Omron Sysmac Studio project 17-701_20171123 (Sysmac Studio 1.19.0.13, StandardProject)

# Controller new_Controller_0: NJ101-1000 version 1.13
Units and slaves: 電源 : NJ-Px3001; CPU : NJ101-1000; 0 : CJ1W-ID211 (J01); 1 : CJ1W-OD211 (J02)
Task PrimaryTask (priority 4, period or condition 2000): prIndexDataChange, prIndex, prError, prSystemInit, prError_S0, prError_S1, prError_S2, prError_S4, prError_S6, prError_S8, prError_S10, prError_S11, prError_S13, prError_S15, prStation1, prStation1_Robot, prStation1_PanelLoad, prStation1_FeedPanelLoad, prStation1_PanelUnLoad, prStation1_FeedPanelUnLoad, prStation2, prStation4, prStation4_TH, prStation4_PanelLoad, prStation4_PanelUnLoad, prStation5, prStation6, prStation7, prStation8, prStation8_CCD, prStation8_ChangeJig, prStation9, prStation10, prStation11, prStation13, prStation15, prStation16, prFeedAndSupplier, prNGCount

TYPE stIndexData : STRUCT
    FinishFlag : ARRAY[0..19] OF BOOL;
    OKFlag : ARRAY[0..19] OF BOOL;
    NGFlag : ARRAY[0..19] OF BOOL;
    ErrorLog : ARRAY[0..19] OF INT;
END_STRUCT END_TYPE

VAR_GLOBAL
    LS_S1_Load_PanelUpDown1Back : BOOL;  (* at ECAT://node#[1,1]/Input Bit 16 bits/Input Bit 00; published *)
    LS_S1_Load_PanelUpDown1Out : BOOL;  (* at ECAT://node#[1,1]/Input Bit 16 bits/Input Bit 01; published *)
    LS_S1_Load_PanelUpDown2Back : BOOL;  (* at ECAT://node#[1,1]/Input Bit 16 bits/Input Bit 02; published *)
    LS_S1_Load_PanelUpDown2Out : BOOL;  (* at ECAT://node#[1,1]/Input Bit 16 bits/Input Bit 03; published *)
    LS_S1_Load_PanelClip1Back : BOOL;  (* at ECAT://node#[1,1]/Input Bit 16 bits/Input Bit 04; published *)
    LS_S1_Load_PanelClip1Out : BOOL;  (* at ECAT://node#[1,1]/Input Bit 16 bits/Input Bit 05; published *)
    LS_S1_Load_PanelClip2Back : BOOL;  (* at ECAT://node#[1,1]/Input Bit 16 bits/Input Bit 06; published *)
    LS_S1_Load_PanelClip2Out : BOOL;  (* at ECAT://node#[1,1]/Input Bit 16 bits/Input Bit 07; published *)
    LS_S1_Load_FixClipBack : BOOL;  (* at ECAT://node#[1,1]/Input Bit 16 bits/Input Bit 08; published *)
    LS_S1_Load_FixClipOut : BOOL;  (* at ECAT://node#[1,1]/Input Bit 16 bits/Input Bit 09; published *)
    LS_S1_Load_AlignmentClipBack : BOOL;  (* at ECAT://node#[1,1]/Input Bit 16 bits/Input Bit 10; published *)
    LS_S1_Load_AlignmentClipOut : BOOL;  (* at ECAT://node#[1,1]/Input Bit 16 bits/Input Bit 11; published *)
    LS_S1_Load_ConveyorClip1Back : BOOL;  (* at ECAT://node#[1,1]/Input Bit 16 bits/Input Bit 12; published *)
    LS_S1_Load_ConveyorClip1Out : BOOL;  (* at ECAT://node#[1,1]/Input Bit 16 bits/Input Bit 13; published *)
    LS_S1_Load_ConveyorClip2Back : BOOL;  (* at ECAT://node#[1,1]/Input Bit 16 bits/Input Bit 14; published *)
    LS_S1_Load_ConveyorClip2Out : BOOL;  (* at ECAT://node#[1,1]/Input Bit 16 bits/Input Bit 15; published *)
    LS_S1_Load_UpDownBack : BOOL;  (* at ECAT://node#[1,2]/Input Bit 16 bits/Input Bit 00; published *)
    LS_S1_Load_UpDownOut : BOOL;  (* at ECAT://node#[1,2]/Input Bit 16 bits/Input Bit 01; published *)
    LS_S1_UnLoad_UpDownBack : BOOL;  (* at ECAT://node#[1,2]/Input Bit 16 bits/Input Bit 02; published *)
    LS_S1_UnLoad_UpDownOut : BOOL;  (* at ECAT://node#[1,2]/Input Bit 16 bits/Input Bit 03; published *)
    LS_S1_UnLoad_ConveyorClip1Back : BOOL;  (* at ECAT://node#[1,2]/Input Bit 16 bits/Input Bit 04; published *)
    LS_S1_UnLoad_ConveyorClip1Out : BOOL;  (* at ECAT://node#[1,2]/Input Bit 16 bits/Input Bit 05; published *)
    LS_S1_UnLoad_ConveyorClip2Back : BOOL;  (* at ECAT://node#[1,2]/Input Bit 16 bits/Input Bit 06; published *)
    LS_S1_UnLoad_ConveyorClip2Out : BOOL;  (* at ECAT://node#[1,2]/Input Bit 16 bits/Input Bit 07; published *)
    LS_S1_UnLoad_FixClipBack : BOOL;  (* at ECAT://node#[1,2]/Input Bit 16 bits/Input Bit 08; published *)
    LS_S1_UnLoad_FixClipOut : BOOL;  (* at ECAT://node#[1,2]/Input Bit 16 bits/Input Bit 09; published *)
    LS_S1_UnLoad_AlignmentClipBack : BOOL;  (* at ECAT://node#[1,2]/Input Bit 16 bits/Input Bit 10; published *)
    LS_S1_UnLoad_AlignmentClipOut : BOOL;  (* at ECAT://node#[1,2]/Input Bit 16 bits/Input Bit 11; published *)
    LS_S1_UnLoad_PanelClip1Back : BOOL;  (* at ECAT://node#[1,2]/Input Bit 16 bits/Input Bit 12; published *)
    LS_S1_UnLoad_PanelClip1Out : BOOL;  (* at ECAT://node#[1,2]/Input Bit 16 bits/Input Bit 13; published *)
    LS_S1_UnLoad_PanelClip2Back : BOOL;  (* at ECAT://node#[1,2]/Input Bit 16 bits/Input Bit 14; published *)
    LS_S1_UnLoad_PanelClip2Out : BOOL;  (* at ECAT://node#[1,2]/Input Bit 16 bits/Input Bit 15; published *)
    LS_S1_UnLoad_PanelUpDown1Back : BOOL;  (* at ECAT://node#[1,3]/Input Bit 16 bits/Input Bit 00; published *)
    LS_S1_UnLoad_PanelUpDown1Out : BOOL;  (* at ECAT://node#[1,3]/Input Bit 16 bits/Input Bit 01; published *)
    LS_S1_UnLoad_PanelUpDown2Back : BOOL;  (* at ECAT://node#[1,3]/Input Bit 16 bits/Input Bit 02; published *)
    LS_S1_UnLoad_PanelUpDown2Out : BOOL;  (* at ECAT://node#[1,3]/Input Bit 16 bits/Input Bit 03; published *)
    SNR_S1_Load_Full : BOOL;  (* 出盤缺盤檢知; at ECAT://node#[1,3]/Input Bit 16 bits/Input Bit 08; published *)
    SNR_S1_UnLoad_Full : BOOL;  (* 收盤滿盤檢知; at ECAT://node#[1,3]/Input Bit 16 bits/Input Bit 09; published *)
    SNR_S1_Load_Feed : BOOL;  (* 下移載出盤檢知; at ECAT://node#[1,3]/Input Bit 16 bits/Input Bit 10; published *)
    SNR_S1_UnLoad_Feed : BOOL;  (* 下移載收盤檢知; at ECAT://node#[1,3]/Input Bit 16 bits/Input Bit 11; published *)
    SNR_S1_Load_PanelFeed : BOOL;  (* 出盤下盤處檢知; at ECAT://node#[1,3]/Input Bit 16 bits/Input Bit 12; published *)
    SNR_S1_Load_PanelClip : BOOL;  (* 出盤夾盤處檢知; at ECAT://node#[1,3]/Input Bit 16 bits/Input Bit 13; published *)
    SNR_S1_UnLoad_PanelFeed : BOOL;  (* 收盤上盤處檢知; at ECAT://node#[1,3]/Input Bit 16 bits/Input Bit 14; published *)
    SNR_S1_UnLoad_PanelClip : BOOL;  (* 收盤夾盤處檢知; at ECAT://node#[1,3]/Input Bit 16 bits/Input Bit 15; published *)
    SOL_S1_Load_PanelUpDown1Back : BOOL;  (* at ECAT://node#[1,4]/Output Bit 16 bits/Output Bit 00; published *)
    SOL_S1_Load_PanelUpDown1Out : BOOL;  (* at ECAT://node#[1,4]/Output Bit 16 bits/Output Bit 01; published *)
    SOL_S1_Load_PanelUpDown2Back : BOOL;  (* at ECAT://node#[1,4]/Output Bit 16 bits/Output Bit 02; published *)
    SOL_S1_Load_PanelUpDown2Out : BOOL;  (* at ECAT://node#[1,4]/Output Bit 16 bits/Output Bit 03; published *)
    SOL_S1_Load_PanelClip : BOOL;  (* at ECAT://node#[1,4]/Output Bit 16 bits/Output Bit 04; published *)
    SOL_S1_Load_FixClip : BOOL;  (* at ECAT://node#[1,4]/Output Bit 16 bits/Output Bit 05; published *)
    SOL_S1_Load_AlignmentClip : BOOL;  (* at ECAT://node#[1,4]/Output Bit 16 bits/Output Bit 06; published *)
    SOL_S1_Load_ConveyorClip : BOOL;  (* at ECAT://node#[1,4]/Output Bit 16 bits/Output Bit 07; published *)
    SOL_S1_Load_UpDown : BOOL;  (* at ECAT://node#[1,4]/Output Bit 16 bits/Output Bit 08; published *)
    RY_S1_Load_FixSpeedMotor : BOOL;  (* at ECAT://node#[1,4]/Output Bit 16 bits/Output Bit 09; published *)
    RY_S1_UnLoad_FixSpeedMotor : BOOL;  (* at ECAT://node#[1,4]/Output Bit 16 bits/Output Bit 10; published *)
    RY_S1_Load_VariableSpeedMotor : BOOL;  (* at ECAT://node#[1,4]/Output Bit 16 bits/Output Bit 11; published *)
    RY_S1_UnLoad_VariableSpeedMotor : BOOL;  (* at ECAT://node#[1,4]/Output Bit 16 bits/Output Bit 12; published *)
    RY_S1_Center_VariableSpeedMotor : BOOL;  (* at ECAT://node#[1,4]/Output Bit 16 bits/Output Bit 13; published *)
    SOL_S1_UnLoad_PanelUpDown1Back : BOOL;  (* at ECAT://node#[1,8]/Output Bit 16 bits/Output Bit 00; published *)
    SOL_S1_UnLoad_PanelUpDown1Out : BOOL;  (* at ECAT://node#[1,8]/Output Bit 16 bits/Output Bit 01; published *)
    SOL_S1_UnLoad_PanelUpDown2Back : BOOL;  (* at ECAT://node#[1,8]/Output Bit 16 bits/Output Bit 02; published *)
    SOL_S1_UnLoad_PanelUpDown2Out : BOOL;  (* at ECAT://node#[1,8]/Output Bit 16 bits/Output Bit 03; published *)
    SOL_S1_UnLoad_PanelClip : BOOL;  (* at ECAT://node#[1,8]/Output Bit 16 bits/Output Bit 04; published *)
    SOL_S1_UnLoad_FixClip : BOOL;  (* at ECAT://node#[1,8]/Output Bit 16 bits/Output Bit 05; published *)
    SOL_S1_UnLoad_AlignmentClip : BOOL;  (* at ECAT://node#[1,8]/Output Bit 16 bits/Output Bit 06; published *)
    SOL_S1_UnLoad_ConveyorClip : BOOL;  (* at ECAT://node#[1,8]/Output Bit 16 bits/Output Bit 07; published *)
    SOL_S1_UnLoad_UpDown : BOOL;  (* at ECAT://node#[1,8]/Output Bit 16 bits/Output Bit 08; published *)
    YAMAHA_Unload_OKStart : BOOL;  (* at ECAT://node#[1,5]/Output Bit 16 bits/Output Bit 00; published *)
    YAMAHA_Unload_NGStart : BOOL;  (* at ECAT://node#[1,5]/Output Bit 16 bits/Output Bit 01; published *)
    YAMAHA_Load_Start : BOOL;  (* at ECAT://node#[1,5]/Output Bit 16 bits/Output Bit 02; published *)
    YAMAHA_UnLoad_Ready : BOOL;  (* at ECAT://node#[1,5]/Output Bit 16 bits/Output Bit 03; published *)
    YAMAHA_Load_Ready : BOOL;  (* at ECAT://node#[1,5]/Output Bit 16 bits/Output Bit 04; published *)
    YAMAHA_Error_SOL_Clip : BOOL;  (* at ECAT://node#[1,6]/Input Bit 16 bits/Input Bit 00; published *)
    YAMAHA_Unload_Finish : BOOL;  (* at ECAT://node#[1,6]/Input Bit 16 bits/Input Bit 01; published *)
    YAMAHA_Load_Finish : BOOL;  (* at ECAT://node#[1,6]/Input Bit 16 bits/Input Bit 02; published *)
    YAMAHA_Unload_ChangePanelStart : BOOL;  (* at ECAT://node#[1,6]/Input Bit 16 bits/Input Bit 03; published *)
    YAMAHA_Load_ChangePanelStart : BOOL;  (* at ECAT://node#[1,6]/Input Bit 16 bits/Input Bit 04; published *)
    YAMAHA_ORG : BOOL;  (* at ECAT://node#[1,6]/Input Bit 16 bits/Input Bit 05; published *)
    YAMAHA_S_Enable : BOOL;  (* at ECAT://node#[1,5]/Output Bit 16 bits/Output Bit 08; published *)
    YAMAHA_S_Control : BOOL;  (* at ECAT://node#[1,5]/Output Bit 16 bits/Output Bit 09; published *)
    YAMAHA_S_Stop : BOOL;  (* at ECAT://node#[1,5]/Output Bit 16 bits/Output Bit 10; published *)
    YAMAHA_S_AutoRun : BOOL;  (* at ECAT://node#[1,5]/Output Bit 16 bits/Output Bit 11; published *)
    YAMAHA_S_INCHome : BOOL;  (* at ECAT://node#[1,5]/Output Bit 16 bits/Output Bit 12; published *)
    YAMAHA_S_ProgramReset : BOOL;  (* at ECAT://node#[1,5]/Output Bit 16 bits/Output Bit 13; published *)
    YAMAHA_S_AlarmReset : BOOL;  (* at ECAT://node#[1,5]/Output Bit 16 bits/Output Bit 14; published *)
    YAMAHA_S_ABSHome : BOOL;  (* at ECAT://node#[1,5]/Output Bit 16 bits/Output Bit 15; published *)
    YAMAHA_S_State_CPUOK : BOOL;  (* at ECAT://node#[1,6]/Input Bit 16 bits/Input Bit 08; published *)
    YAMAHA_S_State_AutoMode : BOOL;  (* at ECAT://node#[1,6]/Input Bit 16 bits/Input Bit 09; published *)
    YAMAHA_S_State_Homed : BOOL;  (* at ECAT://node#[1,6]/Input Bit 16 bits/Input Bit 10; published *)
    YAMAHA_S_State_RobotProgramRun : BOOL;  (* at ECAT://node#[1,6]/Input Bit 16 bits/Input Bit 11; published *)
    YAMAHA_S_State_ProgramReset : BOOL;  (* at ECAT://node#[1,6]/Input Bit 16 bits/Input Bit 12; published *)
    YAMAHA_S_State_Warring : BOOL;  (* at ECAT://node#[1,6]/Input Bit 16 bits/Input Bit 13; published *)
    YAMAHA_S_State_Enable : BOOL;  (* at ECAT://node#[1,6]/Input Bit 16 bits/Input Bit 14; published *)
    YAMAHA_S_State_Alarm : BOOL;  (* at ECAT://node#[1,6]/Input Bit 16 bits/Input Bit 15; published *)
    SNR_S1_Door1 : BOOL;  (* at ECAT://node#[1,3]/Input Bit 16 bits/Input Bit 04; published *)
    SNR_S1_Door2 : BOOL;  (* at ECAT://node#[1,3]/Input Bit 16 bits/Input Bit 05; published *)
    SNR_S1_Door3 : BOOL;  (* at ECAT://node#[1,3]/Input Bit 16 bits/Input Bit 06; published *)
    SNR_S1_Door4 : BOOL;  (* at ECAT://node#[1,3]/Input Bit 16 bits/Input Bit 07; published *)
    LS_S4_Load_PanelUpDown1Back : BOOL;  (* published *)
    LS_S4_Load_PanelUpDown1Out : BOOL;  (* published *)
    LS_S4_Load_PanelUpDown2Back : BOOL;  (* published *)
    LS_S4_Load_PanelUpDown2Out : BOOL;  (* published *)
    LS_S4_Load_PanelClip1Back : BOOL;  (* published *)
    LS_S4_Load_PanelClip1Out : BOOL;  (* published *)
    LS_S4_Load_PanelClip2Back : BOOL;  (* published *)
    LS_S4_Load_PanelClip2Out : BOOL;  (* published *)
    LS_S4_UnLoad_PanelUpDown1Back : BOOL;  (* published *)
    LS_S4_UnLoad_PanelUpDown1Out : BOOL;  (* published *)
    LS_S4_UnLoad_PanelUpDown2Back : BOOL;  (* published *)
    LS_S4_UnLoad_PanelUpDown2Out : BOOL;  (* published *)
    LS_S4_UnLoad_PanelClip1Back : BOOL;  (* published *)
    LS_S4_UnLoad_PanelClip1Out : BOOL;  (* published *)
    LS_S4_UnLoad_PanelClip2Back : BOOL;  (* published *)
    LS_S4_UnLoad_PanelClip2Out : BOOL;  (* published *)
    LS_S4_Center_UpDownBack : BOOL;  (* published *)
    LS_S4_Center_UpDownOut : BOOL;  (* published *)
    LS_S4_Center_ClipBack : BOOL;  (* published *)
    LS_S4_Center_ClipOut : BOOL;  (* published *)
    SNR_S4_Load_Feed : BOOL;  (* published *)
    SNR_S4_UnLoad_Feed : BOOL;  (* published *)
    SNR_S4_Load_Full : BOOL;  (* published *)
    SNR_S4_UnLoad_Full : BOOL;  (* published *)
    SOL_S4_Load_PanelUpDown1Back : BOOL;  (* published *)
    SOL_S4_Load_PanelUpDown1Out : BOOL;  (* published *)
    SOL_S4_Load_PanelUpDown2Back : BOOL;  (* published *)
    SOL_S4_Load_PanelUpDown2Out : BOOL;  (* published *)
    SOL_S4_Load_PanelClip : BOOL;  (* published *)
    SOL_S4_UnLoad_PanelUpDown1Back : BOOL;  (* published *)
    SOL_S4_UnLoad_PanelUpDown1Out : BOOL;  (* published *)
    SOL_S4_UnLoad_PanelUpDown2Back : BOOL;  (* published *)
    SOL_S4_UnLoad_PanelUpDown2Out : BOOL;  (* published *)
    SOL_S4_UnLoad_PanelClip : BOOL;  (* published *)
    SOL_S4_Center_UpDown : BOOL;  (* published *)
    SOL_S4_Center_Clip : BOOL;  (* published *)
    SOL_S2_UpDown : BOOL;  (* published *)
    SOL_S4_MoveBack : BOOL;  (* published *)
    SOL_S4_MoveOut : BOOL;  (* published *)
    SOL_S4_UpDown : BOOL;  (* published *)
    SOL_S4_Clip : BOOL;  (* published *)
    SOL_S4_THMoveBack : BOOL;  (* published *)
    SOL_S4_THMoveOut : BOOL;  (* published *)
    SOL_S6_MoveBack : BOOL;  (* published *)
    SOL_S6_MoveOut : BOOL;  (* published *)
    SOL_S6_UpDown : BOOL;  (* published *)
    SOL_S6_TH : BOOL;  (* published *)
    SOL_S8_MoveBack : BOOL;  (* published *)
    SOL_S8_MoveOut : BOOL;  (* published *)
    SOL_S8_UpDown : BOOL;  (* published *)
    SOL_S8_FixMove : BOOL;  (* published *)
    SOL_S8_Fix : BOOL;  (* published *)
    SOL_S8_TH : BOOL;  (* published *)
    SOL_S8_Turn : BOOL;  (* published *)
    SOL_S8_Clip : BOOL;  (* published *)
    SOL_S10_MoveBack : BOOL;  (* published *)
    SOL_S10_MoveOut : BOOL;  (* published *)
    SOL_S10_UpDown : BOOL;  (* published *)
    SOL_S10_ClipF : BOOL;  (* published *)
    SOL_S10_ClipR : BOOL;  (* published *)
    SOL_S10_TH : BOOL;  (* published *)
    SOL_S10_Turn : BOOL;  (* published *)
    SOL_S11_UpDown : BOOL;  (* published *)
    SOL_S13_UpDown : BOOL;  (* published *)
    SOL_S15_UpDown : BOOL;  (* published *)
    SOL_S6_Vacuum : BOOL;  (* published *)
    SOL_S6_Break : BOOL;  (* published *)
    SOL_S8_VacuumF : BOOL;  (* published *)
    SOL_S8_BreakF : BOOL;  (* published *)
    SOL_S8_VacuumR : BOOL;  (* published *)
    SOL_S8_BreakR : BOOL;  (* published *)
    RY_S6_Full : BOOL;  (* published *)
    RY_S6_Feed : BOOL;  (* published *)
    RY_S8_Full : BOOL;  (* published *)
    RY_S8_Feed : BOOL;  (* published *)
    RY_S10_Full : BOOL;  (* published *)
    RY_S10_Feed : BOOL;  (* published *)
    LS_S2_UpDownBack : BOOL;  (* published *)
    LS_S2_UpDownOut : BOOL;  (* published *)
    LS_S4_MoveBack : BOOL;  (* published *)
    LS_S4_MoveOut : BOOL;  (* published *)
    LS_S4_UpDownBack : BOOL;  (* published *)
    LS_S4_UpDownOut : BOOL;  (* published *)
    LS_S4_ClipBack : BOOL;  (* published *)
    LS_S4_ClipOut : BOOL;  (* published *)
    LS_S4_THMoveBack : BOOL;  (* published *)
    LS_S4_THMoveOut : BOOL;  (* published *)
    LS_S6_MoveBack : BOOL;  (* published *)
    LS_S6_MoveOut : BOOL;  (* published *)
    LS_S6_UpDownBack : BOOL;  (* published *)
    LS_S6_UpDownOut : BOOL;  (* published *)
    LS_S6_THBack : BOOL;  (* published *)
    LS_S6_THOut : BOOL;  (* published *)
    LS_S8_MoveBack : BOOL;  (* published *)
    LS_S8_MoveOut : BOOL;  (* published *)
    LS_S8_UpDownBack : BOOL;  (* published *)
    LS_S8_UpDownOut : BOOL;  (* published *)
    LS_S8_FixMoveBack : BOOL;  (* published *)
    LS_S8_FixMoveOut : BOOL;  (* published *)
    LS_S8_FixBack : BOOL;  (* published *)
    LS_S8_FixOut : BOOL;  (* published *)
    LS_S8_THBack : BOOL;  (* published *)
    LS_S8_THOut : BOOL;  (* published *)
    LS_S8_TurnBack : BOOL;  (* published *)
    LS_S8_TurnOut : BOOL;  (* published *)
    LS_S8_ClipBack : BOOL;  (* published *)
    LS_S8_ClipOut : BOOL;  (* published *)
    LS_S10_MoveBack : BOOL;  (* published *)
    LS_S10_MoveOut : BOOL;  (* published *)
    LS_S10_UpDownBack : BOOL;  (* published *)
    LS_S10_UpDownOut : BOOL;  (* published *)
    LS_S10_ClipFBack : BOOL;  (* published *)
    LS_S10_ClipFOut : BOOL;  (* published *)
    LS_S10_ClipRBack : BOOL;  (* published *)
    LS_S10_ClipROut : BOOL;  (* published *)
    LS_S10_THBack : BOOL;  (* published *)
    LS_S10_THOut : BOOL;  (* published *)
    LS_S10_TurnBack : BOOL;  (* published *)
    LS_S10_TurnOut : BOOL;  (* published *)
    LS_S11_UpDownBack : BOOL;  (* published *)
    LS_S11_UpDownOut : BOOL;  (* published *)
    LS_S13_UpDownBack : BOOL;  (* published *)
    LS_S13_UpDownOut : BOOL;  (* published *)
    LS_S15_UpDownBack : BOOL;  (* published *)
    LS_S15_UpDownOut : BOOL;  (* published *)
    LS_S13_TempHighWarring : BOOL;  (* published *)
    LS_S13_TempLowWarring : BOOL;  (* published *)
    SNR_S4_Feed : BOOL;  (* published *)
    SNR_S5_Check : BOOL;  (* published *)
    SNR_S6_Vacuum : BOOL;  (* published *)
    SNR_S6_Full : BOOL;  (* published *)
    SNR_S6_Feed : BOOL;  (* published *)
    SNR_S7_Check : BOOL;  (* published *)
    SNR_S8_VacuumF : BOOL;  (* published *)
    SNR_S8_VacuumR : BOOL;  (* published *)
    SNR_S8_Full : BOOL;  (* published *)
    SNR_S8_Feed : BOOL;  (* published *)
    SNR_S9_Check : BOOL;  (* published *)
    SNR_S10_Full : BOOL;  (* published *)
    SNR_S10_Feed : BOOL;  (* published *)
    SNR_Index : BOOL;  (* published *)
    SNR_AirSource : BOOL;  (* published *)
    OMRON_FQ2_NG : BOOL;  (* published *)
    OMRON_FQ2_Ready : BOOL;  (* published *)
    OMRON_FQ2_Error : BOOL;  (* published *)
    OMRON_FQ2_Trig : BOOL;  (* published *)
    OMRON_FQ2_IN0 : BOOL;  (* published *)
    OMRON_FQ2_IN1 : BOOL;  (* published *)
    OMRON_FQ2_IN2 : BOOL;  (* published *)
    OMRON_FQ2_IN3 : BOOL;  (* published *)
    OMRON_FQ2_IN4 : BOOL;  (* published *)
    OMRON_FQ2_IN5 : BOOL;  (* published *)
    RY_Index : BOOL;  (* at IOBus://rack#0/slot#1/Ch1_Out/Ch1_Out00; published *)
    BZ : BOOL;  (* at IOBus://rack#0/slot#1/Ch1_Out/Ch1_Out04; published *)
    YL : BOOL;  (* at IOBus://rack#0/slot#1/Ch1_Out/Ch1_Out02; published *)
    GL : BOOL;  (* at IOBus://rack#0/slot#1/Ch1_Out/Ch1_Out03; published *)
    RL : BOOL;  (* at IOBus://rack#0/slot#1/Ch1_Out/Ch1_Out01; published *)
    Invertor_Ready : BOOL;  (* at IOBus://rack#0/slot#0/Ch1_In/Ch1_In03; published *)
    PB_Start : BOOL;  (* at IOBus://rack#0/slot#0/Ch1_In/Ch1_In00; published *)
    PB_Reset : BOOL;  (* at IOBus://rack#0/slot#0/Ch1_In/Ch1_In01; published *)
    PB_EStop : BOOL;  (* at IOBus://rack#0/slot#0/Ch1_In/Ch1_In02; published *)
    HMIPB_SOL_S1_Load_PanelUpDown1Back : BOOL;  (* published *)
    HMIPB_SOL_S1_Load_PanelUpDown1Out : BOOL;  (* published *)
    HMIPB_SOL_S1_Load_PanelUpDown2Back : BOOL;  (* published *)
    HMIPB_SOL_S1_Load_PanelUpDown2Out : BOOL;  (* published *)
    HMIPB_SOL_S1_Load_PanelClip : BOOL;  (* published *)
    HMIPB_SOL_S1_Load_FixClip : BOOL;  (* published *)
    HMIPB_SOL_S1_Load_AlignmentClip : BOOL;  (* published *)
    HMIPB_SOL_S1_Load_ConveyorClip : BOOL;  (* published *)
    HMIPB_SOL_S1_Load_UpDown : BOOL;  (* published *)
    HMIPB_RY_S1_Load_FixSpeedMotor : BOOL;  (* published *)
    HMIPB_RY_S1_UnLoad_FixSpeedMotor : BOOL;  (* published *)
    HMIPB_RY_S1_Load_VariableSpeedMotor : BOOL;  (* published *)
    HMIPB_RY_S1_UnLoad_VariableSpeedMotor : BOOL;  (* published *)
    HMIPB_RY_S1_Center_VariableSpeedMotor : BOOL;  (* published *)
    HMIPB_SOL_S1_UnLoad_PanelUpDown1Back : BOOL;  (* published *)
    HMIPB_SOL_S1_UnLoad_PanelUpDown1Out : BOOL;  (* published *)
    HMIPB_SOL_S1_UnLoad_PanelUpDown2Back : BOOL;  (* published *)
    HMIPB_SOL_S1_UnLoad_PanelUpDown2Out : BOOL;  (* published *)
    HMIPB_SOL_S1_UnLoad_PanelClip : BOOL;  (* published *)
    HMIPB_SOL_S1_UnLoad_FixClip : BOOL;  (* published *)
    HMIPB_SOL_S1_UnLoad_AlignmentClip : BOOL;  (* published *)
    HMIPB_SOL_S1_UnLoad_ConveyorClip : BOOL;  (* published *)
    HMIPB_SOL_S1_UnLoad_UpDown : BOOL;  (* published *)
    HMIPB_YAMAHA_Unload_OKStart : BOOL;  (* published *)
    HMIPB_YAMAHA_Unload_NGStart : BOOL;  (* published *)
    HMIPB_YAMAHA_Load_Start : BOOL;  (* published *)
    HMIPB_YAMAHA_UnLoad_Ready : BOOL;  (* published *)
    HMIPB_YAMAHA_Load_Ready : BOOL;  (* published *)
    HMIPB_YAMAHA_Unload_ChangePanelStart : BOOL;  (* published *)
    HMIPB_YAMAHA_Load_ChangePanelStart : BOOL;  (* published *)
    HMIPB_YAMAHA_ORG : BOOL;  (* published *)
    HMIPB_YAMAHA_S_Enable : BOOL;  (* published *)
    HMIPB_YAMAHA_S_Control : BOOL;  (* published *)
END_VAR
VAR_GLOBAL RETAIN
    HMIPB_YAMAHA_S_Stop : BOOL;  (* published *)
END_VAR
VAR_GLOBAL
    HMIPB_YAMAHA_S_AutoRun : BOOL;  (* published *)
    HMIPB_YAMAHA_S_INCHome : BOOL;  (* published *)
    HMIPB_YAMAHA_S_ProgramReset : BOOL;  (* published *)
    HMIPB_YAMAHA_S_AlarmReset : BOOL;  (* published *)
    HMIPB_YAMAHA_S_ABSHome : BOOL;  (* published *)
    HMIPB_SOL_S4_Load_PanelUpDown1Back : BOOL;  (* published *)
    HMIPB_SOL_S4_Load_PanelUpDown1Out : BOOL;  (* published *)
    HMIPB_SOL_S4_Load_PanelUpDown2Back : BOOL;  (* published *)
    HMIPB_SOL_S4_Load_PanelUpDown2Out : BOOL;  (* published *)
    HMIPB_SOL_S4_Load_PanelClip : BOOL;  (* published *)
    HMIPB_SOL_S4_UnLoad_PanelUpDown1Back : BOOL;  (* published *)
    HMIPB_SOL_S4_UnLoad_PanelUpDown1Out : BOOL;  (* published *)
    HMIPB_SOL_S4_UnLoad_PanelUpDown2Back : BOOL;  (* published *)
    HMIPB_SOL_S4_UnLoad_PanelUpDown2Out : BOOL;  (* published *)
    HMIPB_SOL_S4_UnLoad_PanelClip : BOOL;  (* published *)
    HMIPB_SOL_S4_Center_UpDown : BOOL;  (* published *)
    HMIPB_SOL_S4_Center_Clip : BOOL;  (* published *)
    HMIPB_SOL_S2_UpDown : BOOL;  (* published *)
    HMIPB_SOL_S4_MoveBack : BOOL;  (* published *)
    HMIPB_SOL_S4_MoveOut : BOOL;  (* published *)
    HMIPB_SOL_S4_UpDown : BOOL;  (* published *)
    HMIPB_SOL_S4_Clip : BOOL;  (* published *)
    HMIPB_SOL_S4_THMoveBack : BOOL;  (* published *)
    HMIPB_SOL_S4_THMoveOut : BOOL;  (* published *)
    HMIPB_SOL_S6_MoveBack : BOOL;  (* published *)
    HMIPB_SOL_S6_MoveOut : BOOL;  (* published *)
    HMIPB_SOL_S6_UpDown : BOOL;  (* published *)
    HMIPB_SOL_S6_TH : BOOL;  (* published *)
    HMIPB_SOL_S8_MoveBack : BOOL;  (* published *)
    HMIPB_SOL_S8_MoveOut : BOOL;  (* published *)
    HMIPB_SOL_S8_UpDown : BOOL;  (* published *)
    HMIPB_SOL_S8_FixMove : BOOL;  (* published *)
    HMIPB_SOL_S8_Fix : BOOL;  (* published *)
    HMIPB_SOL_S8_TH : BOOL;  (* published *)
    HMIPB_SOL_S8_Turn : BOOL;  (* published *)
    HMIPB_SOL_S8_Clip : BOOL;  (* published *)
    HMIPB_SOL_S10_MoveBack : BOOL;  (* published *)
    HMIPB_SOL_S10_MoveOut : BOOL;  (* published *)
    HMIPB_SOL_S10_UpDown : BOOL;  (* published *)
    HMIPB_SOL_S10_ClipF : BOOL;  (* published *)
    HMIPB_SOL_S10_ClipR : BOOL;  (* published *)
    HMIPB_SOL_S10_TH : BOOL;  (* published *)
    HMIPB_SOL_S10_Turn : BOOL;  (* published *)
    HMIPB_SOL_S11_UpDown : BOOL;  (* published *)
    HMIPB_SOL_S13_UpDown : BOOL;  (* published *)
    HMIPB_SOL_S15_UpDown : BOOL;  (* published *)
    HMIPB_SOL_S6_Vacuum : BOOL;  (* published *)
    HMIPB_SOL_S6_Break : BOOL;  (* published *)
    HMIPB_SOL_S8_VacuumF : BOOL;  (* published *)
    HMIPB_SOL_S8_BreakF : BOOL;  (* published *)
    HMIPB_SOL_S8_VacuumR : BOOL;  (* published *)
    HMIPB_SOL_S8_BreakR : BOOL;  (* published *)
    HMIPB_RY_S6_Full : BOOL;  (* published *)
    HMIPB_RY_S6_Feed : BOOL;  (* published *)
    HMIPB_RY_S8_Full : BOOL;  (* published *)
    HMIPB_RY_S8_Feed : BOOL;  (* published *)
    HMIPB_RY_S10_Full : BOOL;  (* published *)
    HMIPB_RY_S10_Feed : BOOL;  (* published *)
    HMIPB_OMRON_FQ2_Trig : BOOL;  (* published *)
    HMIPB_RY_Index : BOOL;  (* published *)
    HMIPB_PB_Start : BOOL;  (* published *)
    HMIPB_PB_Reset : BOOL;  (* published *)
    HMIPB_S11_StandarValueSet : BOOL;  (* published *)
    HMIPB_S15_StandarValueSet : BOOL;  (* published *)
    DisablePB : ARRAY[0..19] OF BOOL;  (* published *)
    TestPB : ARRAY[0..19] OF BOOL;  (* published *)
    Error_LS_S1_Load_PanelUpDown1Back : BOOL;  (* published *)
    Error_LS_S1_Load_PanelUpDown1Out : BOOL;  (* published *)
    Error_LS_S1_Load_PanelUpDown2Back : BOOL;  (* published *)
    Error_LS_S1_Load_PanelUpDown2Out : BOOL;  (* published *)
    Error_LS_S1_Load_PanelClip1Back : BOOL;  (* published *)
    Error_LS_S1_Load_PanelClip1Out : BOOL;  (* published *)
    Error_LS_S1_Load_PanelClip2Back : BOOL;  (* published *)
    Error_LS_S1_Load_PanelClip2Out : BOOL;  (* published *)
    Error_LS_S1_Load_FixClipBack : BOOL;  (* published *)
    Error_LS_S1_Load_FixClipOut : BOOL;  (* published *)
    Error_LS_S1_Load_AlignmentClipBack : BOOL;  (* published *)
    Error_LS_S1_Load_AlignmentClipOut : BOOL;  (* published *)
    Error_LS_S1_Load_ConveyorClip1Back : BOOL;  (* published *)
    Error_LS_S1_Load_ConveyorClip1Out : BOOL;  (* published *)
    Error_LS_S1_Load_ConveyorClip2Back : BOOL;  (* published *)
    Error_LS_S1_Load_ConveyorClip2Out : BOOL;  (* published *)
    Error_LS_S1_Load_UpDownBack : BOOL;  (* published *)
    Error_LS_S1_Load_UpDownOut : BOOL;  (* published *)
    Error_LS_S1_UnLoad_UpDownBack : BOOL;  (* published *)
    Error_LS_S1_UnLoad_UpDownOut : BOOL;  (* published *)
    Error_LS_S1_UnLoad_ConveyorClip1Back : BOOL;  (* published *)
    Error_LS_S1_UnLoad_ConveyorClip1Out : BOOL;  (* published *)
    Error_LS_S1_UnLoad_ConveyorClip2Back : BOOL;  (* published *)
    Error_LS_S1_UnLoad_ConveyorClip2Out : BOOL;  (* published *)
    Error_LS_S1_UnLoad_FixClipBack : BOOL;  (* published *)
    Error_LS_S1_UnLoad_FixClipOut : BOOL;  (* published *)
    Error_LS_S1_UnLoad_AlignmentClipBack : BOOL;  (* published *)
    Error_LS_S1_UnLoad_AlignmentClipOut : BOOL;  (* published *)
    Error_LS_S1_UnLoad_PanelClip1Back : BOOL;  (* published *)
    Error_LS_S1_UnLoad_PanelClip1Out : BOOL;  (* published *)
    Error_LS_S1_UnLoad_PanelClip2Back : BOOL;  (* published *)
    Error_LS_S1_UnLoad_PanelClip2Out : BOOL;  (* published *)
    Error_LS_S1_UnLoad_PanelUpDown1Back : BOOL;  (* published *)
    Error_LS_S1_UnLoad_PanelUpDown1Out : BOOL;  (* published *)
    Error_LS_S1_UnLoad_PanelUpDown2Back : BOOL;  (* published *)
    Error_LS_S1_UnLoad_PanelUpDown2Out : BOOL;  (* published *)
    Error_SNR_S1_Load_Full : BOOL;  (* published *)
    Error_SNR_S1_UnLoad_Full : BOOL;  (* published *)
    Error_SNR_S1_Load_Feed : BOOL;  (* published *)
    Error_SNR_S1_UnLoad_Feed : BOOL;  (* published *)
    Error_SNR_S1_Load_PanelFeed : BOOL;  (* published *)
    Error_SNR_S1_Load_PanelClip : BOOL;  (* published *)
    Error_SNR_S1_UnLoad_PanelFeed : BOOL;  (* published *)
    Error_SNR_S1_UnLoad_PanelClip : BOOL;  (* published *)
    Error_YAMAHA_Error_SOL_Clip : BOOL;  (* published *)
    Error_YAMAHA_S_State_Warring : BOOL;  (* published *)
    Error_YAMAHA_S_State_Alarm : BOOL;  (* published *)
    Error_LS_S4_Load_PanelUpDown1Back : BOOL;  (* published *)
    Error_LS_S4_Load_PanelUpDown1Out : BOOL;  (* published *)
    Error_LS_S4_Load_PanelUpDown2Back : BOOL;  (* published *)
    Error_LS_S4_Load_PanelUpDown2Out : BOOL;  (* published *)
    Error_LS_S4_Load_PanelClip1Back : BOOL;  (* published *)
    Error_LS_S4_Load_PanelClip1Out : BOOL;  (* published *)
    Error_LS_S4_Load_PanelClip2Back : BOOL;  (* published *)
    Error_LS_S4_Load_PanelClip2Out : BOOL;  (* published *)
    Error_LS_S4_UnLoad_PanelUpDown1Back : BOOL;  (* published *)
    Error_LS_S4_UnLoad_PanelUpDown1Out : BOOL;  (* published *)
    Error_LS_S4_UnLoad_PanelUpDown2Back : BOOL;  (* published *)
    Error_LS_S4_UnLoad_PanelUpDown2Out : BOOL;  (* published *)
    Error_LS_S4_UnLoad_PanelClip1Back : BOOL;  (* published *)
    Error_LS_S4_UnLoad_PanelClip1Out : BOOL;  (* published *)
    Error_LS_S4_UnLoad_PanelClip2Back : BOOL;  (* published *)
    Error_LS_S4_UnLoad_PanelClip2Out : BOOL;  (* published *)
    Error_LS_S4_Center_UpDownBack : BOOL;  (* published *)
    Error_LS_S4_Center_UpDownOut : BOOL;  (* published *)
    Error_LS_S4_Center_ClipBack : BOOL;  (* published *)
    Error_LS_S4_Center_ClipOut : BOOL;  (* published *)
    Error_SNR_S4_Load_Feed : BOOL;  (* published *)
    Error_SNR_S4_UnLoad_Feed : BOOL;  (* published *)
    Error_SNR_S4_Load_Full : BOOL;  (* published *)
    Error_SNR_S4_UnLoad_Full : BOOL;  (* published *)
    Error_LS_S2_UpDownBack : BOOL;  (* published *)
    Error_LS_S2_UpDownOut : BOOL;  (* published *)
    Error_LS_S2_UpDownOut1 : BOOL;  (* published *)
    Error_LS_S4_MoveBack : BOOL;  (* published *)
    Error_LS_S4_MoveOut : BOOL;  (* published *)
    Error_LS_S4_UpDownBack : BOOL;  (* published *)
    Error_LS_S4_UpDownOut : BOOL;  (* published *)
    Error_LS_S4_UpDownOut1 : BOOL;  (* published *)
    Error_LS_S4_ClipBack : BOOL;  (* published *)
    Error_LS_S4_ClipOut : BOOL;  (* published *)
    Error_LS_S4_THMoveBack : BOOL;  (* published *)
    Error_LS_S4_THMoveOut : BOOL;  (* published *)
    Error_LS_S6_MoveBack : BOOL;  (* published *)
    Error_LS_S6_MoveOut : BOOL;  (* published *)
    Error_LS_S6_UpDownBack : BOOL;  (* published *)
    Error_LS_S6_UpDownOut : BOOL;  (* published *)
    Error_LS_S6_UpDownOut1 : BOOL;  (* published *)
    Error_LS_S6_THBack : BOOL;  (* published *)
    Error_LS_S6_THOut : BOOL;  (* published *)
    Error_LS_S8_MoveBack : BOOL;  (* published *)
    Error_LS_S8_MoveOut : BOOL;  (* published *)
    Error_LS_S8_UpDownBack : BOOL;  (* published *)
    Error_LS_S8_UpDownOut : BOOL;  (* published *)
    Error_LS_S8_UpDownOut1 : BOOL;  (* published *)
    Error_LS_S8_FixMoveBack : BOOL;  (* published *)
    Error_LS_S8_FixMoveOut : BOOL;  (* published *)
    Error_LS_S8_FixBack : BOOL;  (* published *)
    Error_LS_S8_FixOut : BOOL;  (* published *)
    Error_LS_S8_THBack : BOOL;  (* published *)
    Error_LS_S8_THOut : BOOL;  (* published *)
    Error_LS_S8_TurnBack : BOOL;  (* published *)
    Error_LS_S8_TurnOut : BOOL;  (* published *)
    Error_LS_S8_ClipBack : BOOL;  (* published *)
    Error_LS_S8_ClipOut : BOOL;  (* published *)
    Error_LS_S10_MoveBack : BOOL;  (* published *)
    Error_LS_S10_MoveOut : BOOL;  (* published *)
    Error_LS_S10_UpDownBack : BOOL;  (* published *)
    Error_LS_S10_UpDownOut : BOOL;  (* published *)
    Error_LS_S10_UpDownOut1 : BOOL;  (* published *)
    Error_LS_S10_ClipFBack : BOOL;  (* published *)
    Error_LS_S10_ClipFOut : BOOL;  (* published *)
    Error_LS_S10_ClipRBack : BOOL;  (* published *)
    Error_LS_S10_ClipROut : BOOL;  (* published *)
    Error_LS_S10_THBack : BOOL;  (* published *)
    Error_LS_S10_THOut : BOOL;  (* published *)
    Error_LS_S10_TurnBack : BOOL;  (* published *)
    Error_LS_S10_TurnOut : BOOL;  (* published *)
    Error_LS_S11_UpDownBack : BOOL;  (* published *)
    Error_LS_S11_UpDownOut : BOOL;  (* published *)
    Error_LS_S11_UpDownOut1 : BOOL;  (* published *)
    Error_LS_S13_UpDownBack : BOOL;  (* published *)
    Error_LS_S13_UpDownOut : BOOL;  (* published *)
    Error_LS_S13_UpDownOut1 : BOOL;  (* published *)
    Error_LS_S15_UpDownBack : BOOL;  (* published *)
    Error_LS_S15_UpDownOut : BOOL;  (* published *)
    Error_LS_S15_UpDownOut1 : BOOL;  (* published *)
    Error_LS_S13_TempHighWarring : BOOL;  (* published *)
    Error_LS_S13_TempLowWarring : BOOL;  (* published *)
    Error_SNR_S4_Feed : BOOL;  (* published *)
    Error_SNR_S5_Check : BOOL;  (* published *)
    Error_SNR_S6_Vacuum : BOOL;  (* published *)
    Error_SNR_S6_Full : BOOL;  (* published *)
    Error_SNR_S6_Feed : BOOL;  (* published *)
    Error_SNR_S7_Check : BOOL;  (* published *)
    Error_SNR_S8_VacuumF : BOOL;  (* published *)
    Error_SNR_S8_VacuumR : BOOL;  (* published *)
    Error_SNR_S8_Full : BOOL;  (* published *)
    Error_SNR_S8_Feed : BOOL;  (* published *)
    Error_SNR_S9_Check : BOOL;  (* published *)
    Error_SNR_S10_Full : BOOL;  (* published *)
    Error_SNR_S10_Feed : BOOL;  (* published *)
    Error_SNR_Index : BOOL;  (* published *)
    Error_SNR_AirSource : BOOL;  (* published *)
    Error_OMRON_FQ2_Error : BOOL;  (* published *)
    Error_Invertor_Ready : BOOL;  (* published *)
    Error_PB_EStop : BOOL;  (* published *)
    Error_LS_Door : BOOL;  (* published *)
    Error_NGCount : ARRAY[0..19] OF BOOL;  (* published *)
    AutoStatus : BOOL;  (* published *)
    SystemReadyStatus : BOOL;  (* published *)
    MachineRunStatus : BOOL;  (* published *)
    StepMode : BOOL;  (* published *)
    Manual2AutoFlag : BOOL;
    FeedStart_S4_Load : BOOL;
    FeedFinish_S4_Load : BOOL;
    FeedStart_S4_UnLoad : BOOL;
    FeedFinish_S4_UnLoad : BOOL;
    CCDStartFlag : BOOL;
    CCDFinishFlag : BOOL;
    CCD_Check_NG : BOOL;
END_VAR
VAR_GLOBAL RETAIN
    S8_ChangeJigStartFlag : BOOL;
END_VAR
VAR_GLOBAL
    FeedStart : ARRAY[0..19] OF BOOL;
    FeedFinish : ARRAY[0..19] OF BOOL;
    ErrorStatus : ARRAY[0..19] OF BOOL;
    ErrorStatus_TH : ARRAY[0..19] OF BOOL;
    MappingOK : ARRAY[0..19] OF BOOL;  (* published *)
    MappingNG : ARRAY[0..19] OF BOOL;  (* published *)
    ErrorStatus_S1_Load : BOOL;
    ErrorStatus_S1_FeedPanelLoad : BOOL;
    ErrorStatus_S1_UnLoad : BOOL;
    ErrorStatus_S1_FeedPanelUnLoad : BOOL;
    ErrorStatus_S1_Center : BOOL;
    ErrorStatus_S4_Load : BOOL;
    ErrorStatus_S4_UnLoad : BOOL;
    ErrorStatus_S4_Center : BOOL;
    ErrorStatus_S8_Fix : BOOL;
    ErrorStatus_MachineStop : BOOL;
    ErrorStatus_MachineStop_Record : BOOL;
    ErrorStatus_MachineNonStop : BOOL;
END_VAR
VAR_GLOBAL RETAIN
    IndexData : ARRAY[0..19] OF stIndexData;  (* published *)
    BatchIndexCount : DINT;  (* published *)
    BatchOKCount : DINT;  (* published *)
    BatchNGCount : DINT;  (* published *)
    BatchTargetCount : DINT;  (* published *)
    HMISV_Index_DelayTime : DINT;  (* published *)
END_VAR
VAR_GLOBAL
    HMIPV_S11_CurrentValue : DINT;  (* published *)
END_VAR
VAR_GLOBAL RETAIN
    HMISV_S11_StandarValue : DINT;  (* published *)
    HMISV_S11_MaxValue : DINT;  (* published *)
    HMISV_S11_MinValue : DINT;  (* published *)
    HMISV_S11_PValue : DINT;  (* published *)
    HMISV_S11_NValue : DINT;  (* published *)
    HMISV_S13_PressTime : DINT;  (* published *)
END_VAR
VAR_GLOBAL
    HMIPV_S15_CurrentValue : DINT;  (* published *)
END_VAR
VAR_GLOBAL RETAIN
    HMISV_S15_StandarValue : DINT;  (* published *)
    HMISV_S15_MaxValue : DINT;  (* published *)
    HMISV_S15_MinValue : DINT;  (* published *)
    HMISV_S15_PValue : DINT;  (* published *)
    HMISV_S15_NValue : DINT;  (* published *)
    FullNotExistTime : ARRAY[0..19] OF DINT;  (* published *)
    FullExistTime : ARRAY[0..19] OF DINT;  (* published *)
    FullNotExistErrorTime : ARRAY[0..19] OF DINT;  (* published *)
    FeedNotExistTime : ARRAY[0..19] OF DINT;  (* published *)
    FeedExistTime : ARRAY[0..19] OF DINT;  (* published *)
    CycleTime : ARRAY[0..19] OF DINT;  (* published *)
    CurrentCycleTime : ARRAY[0..9] OF DINT;  (* published *)
    AverageCycleTime : DINT;  (* published *)
END_VAR

PROGRAM prSystemInit
VAR
    SystemInitFlow : INT := 0;
    TON1 : TON;
    TON2 : TON;
    TON3 : TON;
    TON_3 : TON;
    R_TRIG_3 : R_TRIG;
    R_TRIG_4 : R_TRIG;
    Flash_1S_1S : BOOL;
END_VAR
VAR_EXTERNAL
    AutoStatus : BOOL;
    SystemReadyStatus : BOOL;
    PB_EStop : BOOL;
    Error_PB_EStop : BOOL;
    Manual2AutoFlag : BOOL;
    ErrorStatus_MachineStop : BOOL;
    ErrorStatus_MachineNonStop : BOOL;
    ErrorStatus_MachineStop_Record : BOOL;
    BZ : BOOL;
    RL : BOOL;
    GL : BOOL;
    YL : BOOL;
    MappingOK : ARRAY[0..19] OF BOOL;
    IndexData : ARRAY[0..19] OF stIndexData;
    MappingNG : ARRAY[0..19] OF BOOL;
    PB_Start : BOOL;
    HMIPB_PB_Start : BOOL;
    PB_Reset : BOOL;
    HMIPB_PB_Reset : BOOL;
    MachineRunStatus : BOOL;
    BatchOKCount : DINT;
    BatchTargetCount : DINT;
    BatchIndexCount : DINT;
    DisablePB : ARRAY[0..19] OF BOOL;
    Error_LS_Door : BOOL;
    SNR_S1_Door1 : BOOL;
    SNR_S1_Door2 : BOOL;
    SNR_S1_Door3 : BOOL;
    SNR_S1_Door4 : BOOL;
    StepMode : BOOL;
END_VAR
(******************************************************************
程式:系統初始化
作者:蔡相偉
版本資訊:1.0.0		2016/5/26

全部狀態RESET=0
伺服上電=1
伺服未回HOME=2
伺服Servo on=3
伺服Ready=4
夾爪回=5
夾爪前後回=6
伺服上下軸Serch Home=7
伺服上下軸Serch Home中=8
伺服上下軸Serch Home完成=9
伺服橫移軸Serch Home=10
伺服橫移軸Serch Home中=11
伺服橫移軸Serch Home完成=12
自動SET=13
系統READY SET=14
Init完成=15
******************************************************************)
//全部狀態RESET=0
IF P_First_Run THEN
	SystemInitFlow:=0;
	AutoStatus:=FALSE;
	SystemReadyStatus:=FALSE;
END_IF;

//伺服上電=1
IF SystemInitFlow=0 AND P_Off AND PB_EStop AND NOT(Error_PB_EStop) AND NOT(AutoStatus) AND NOT(SystemReadyStatus) (*AND MC_Axis000.DrvStatus.MainPower AND MC_Axis001.DrvStatus.MainPower*) THEN
	SystemInitFlow:=1;
END_IF;

//伺服未回HOME=2
IF SystemInitFlow=1 (*AND (NOT(MC_Axis000.Details.Homed) OR NOT(MC_Axis001.Details.Homed))*) THEN
	SystemInitFlow:=2;
END_IF;

//伺服Servo on=3
IF SystemInitFlow=2 THEN
	SystemInitFlow:=3;
END_IF;
IF SystemInitFlow=3 THEN
	//PB_ServoOn_UpDown:=TRUE;
	//PB_ServoOn_Move:=TRUE;
	;
END_IF;

//伺服Ready=4
IF SystemInitFlow=3 (*AND AxMove.bServoOn AND AxUpDown.bServoOn AND MC_Axis000.DrvStatus.Ready AND MC_Axis001.DrvStatus.Ready*) THEN
	SystemInitFlow:=4;
END_IF;

//夾爪回=5
TON1(In:=SystemInitFlow=4 , PT:=t#1s);
IF SystemInitFlow=4 AND TON1.Q THEN
	SystemInitFlow:=5;
END_IF;
IF SystemInitFlow=5 THEN
	;
END_IF;

//夾爪前後回=6
IF SystemInitFlow=5 THEN
	SystemInitFlow:=6;
END_IF;
IF SystemInitFlow=6 THEN
	//SOL_Move:=FALSE;
	;
END_IF;

//伺服上下軸Serch Home=7
IF SystemInitFlow=6  THEN
	SystemInitFlow:=7;
END_IF;
IF SystemInitFlow=7 THEN
	//AxUpDown.pbSerchHome:=TRUE;
	;
END_IF;

//伺服上下軸Serch Home中=8
IF SystemInitFlow=7 THEN
	//AxUpDown.pbSerchHome:=FALSE;
	SystemInitFlow:=8;
END_IF;

//伺服上下軸Serch Home完成=9
IF SystemInitFlow=8  THEN
	SystemInitFlow:=9;
END_IF;

//伺服橫移軸Serch Home=10
IF SystemInitFlow=9  THEN
	SystemInitFlow:=10;
END_IF;
IF SystemInitFlow=10 THEN
	//AxMove.pbSerchHome:=TRUE;
	;
END_IF;

//伺服橫移軸Serch Home中=11
IF SystemInitFlow=10 THEN
	//AxMove.pbSerchHome:=FALSE;
	SystemInitFlow:=11;
END_IF;

//伺服橫移軸Serch Home完成=12
IF SystemInitFlow=11 THEN
	SystemInitFlow:=12;
END_IF;

//自動SET=13
IF SystemInitFlow=12  THEN
	SystemInitFlow:=13;
END_IF;
IF SystemInitFlow=13 THEN
	AutoStatus:=TRUE;
END_IF;

//系統READY SET=14
IF SystemInitFlow=13 AND AutoStatus THEN
	SystemInitFlow:=14;
END_IF;
IF SystemInitFlow=14 THEN
	SystemReadyStatus:=TRUE;
END_IF;

//Init完成=15
IF SystemInitFlow=14 AND SystemReadyStatus THEN
	SystemInitFlow:=15;
END_IF;
//******************************************************************
//全自動起動
R_TRIG_4(CLK:= PB_Start OR HMIPB_PB_Start);
IF AutoStatus AND NOT(PB_Reset OR HMIPB_PB_Reset OR NOT(PB_Estop) OR ErrorStatus_MachineStop OR Error_LS_Door OR BatchOKCount>=BatchTargetCount) AND
	R_TRIG_4.Q THEN
	MachineRunStatus:=TRUE;
	StepMode:=FALSE;
END_IF;
//停止
IF PB_Reset OR HMIPB_PB_Reset OR NOT(PB_Estop) OR ErrorStatus_MachineStop OR Error_LS_Door OR BatchOKCount>=BatchTargetCount THEN
	MachineRunStatus:=FALSE;
END_IF;
//門開啟設備暫停
IF NOT(SNR_S1_Door1 AND SNR_S1_Door2 AND SNR_S1_Door3 AND SNR_S1_Door4) THEN
	StepMode:=TRUE;
END_IF;
//產能到達關閉第1站
IF BatchIndexCount+BatchOKCount>=BatchTargetCount THEN
	DisablePB[1]:=TRUE;
ELSE
	DisablePB[1]:=FALSE;
END_IF;
//******************************************************************
//手動轉自動
R_TRIG_3(CLK:= AutoStatus ,Q=> Manual2AutoFlag );
(******************************************************************
程式:燈號及蜂鳴器
作者:蔡相偉
版本資訊:1.0.0		2016/5/26
******************************************************************)
//BZ停止
TON_3(IN:=(ErrorStatus_MachineStop OR ErrorStatus_MachineNonStop OR ErrorStatus_MachineStop_Record) , PT:=t#10s);
//BZ
IF (ErrorStatus_MachineStop OR ErrorStatus_MachineNonStop OR ErrorStatus_MachineStop_Record) AND NOT(TON_3.Q) THEN
	BZ:=Flash_1S_1S;
	ELSE
	BZ:=FALSE;
END_IF;
//紅燈
IF ErrorStatus_MachineStop OR ErrorStatus_MachineStop_Record THEN
	RL:=TRUE;
	ELSE
	RL:=FALSE;
END_IF;
//綠燈
IF NOT(ErrorStatus_MachineStop) AND
	NOT(ErrorStatus_MachineNonStop) AND NOT(ErrorStatus_MachineStop_Record) THEN
	GL:=TRUE;
	ELSE
	GL:=FALSE;
END_IF;
//黃燈
IF ErrorStatus_MachineNonStop THEN
	YL:=TRUE;
	ELSE
	YL:=FALSE;
END_IF;

//**************************************************************************************************
//Mapping
MappingOK[1]:=IndexData[1].OKFlag[1];
MappingOK[2]:=IndexData[2].OKFlag[2];
MappingOK[4]:=IndexData[4].OKFlag[4];
MappingOK[5]:=IndexData[5].OKFlag[5];
MappingOK[6]:=IndexData[6].OKFlag[6];
MappingOK[7]:=IndexData[7].OKFlag[7];
MappingOK[8]:=IndexData[8].OKFlag[8];
MappingOK[9]:=IndexData[9].OKFlag[9];
MappingOK[10]:=IndexData[10].OKFlag[10];
MappingOK[11]:=IndexData[11].OKFlag[11];
MappingOK[13]:=IndexData[13].OKFlag[13];
MappingOK[15]:=IndexData[15].OKFlag[15];
MappingOK[16]:=IndexData[16].OKFlag[16];
MappingNG[1]:=IndexData[1].NGFlag[1];
MappingNG[2]:=IndexData[2].NGFlag[2];
MappingNG[4]:=IndexData[4].NGFlag[4];
MappingNG[5]:=IndexData[5].NGFlag[5];
MappingNG[6]:=IndexData[6].NGFlag[6];
MappingNG[7]:=IndexData[7].NGFlag[7];
MappingNG[8]:=IndexData[8].NGFlag[8];
MappingNG[9]:=IndexData[9].NGFlag[9];
MappingNG[10]:=IndexData[10].NGFlag[10];
MappingNG[11]:=IndexData[11].NGFlag[11];
MappingNG[13]:=IndexData[13].NGFlag[13];
MappingNG[15]:=IndexData[15].NGFlag[15];
MappingNG[16]:=IndexData[16].NGFlag[16];
//**************************************************************************************************
//Flash_1sOn_1sOff
TON2(In:=NOT(Flash_1S_1S), PT:=t#1s);
TON3(In:=(Flash_1S_1S), PT:=t#1s);
IF TON2.Q THEN
	Flash_1S_1S:=TRUE;
END_IF;
IF TON3.Q THEN
	Flash_1S_1S:=FALSE;
END_IF;
END_PROGRAM

PROGRAM prIndexDataChange
VAR
    R_TRIG_1 : R_TRIG;
END_VAR
VAR_EXTERNAL
    SNR_Index : BOOL;
    IndexData : ARRAY[0..19] OF stIndexData;
    SystemReadyStatus : BOOL;
END_VAR
(*本機轉盤*)
R_TRIG_1(CLK:=SNR_Index);
IF SystemReadyStatus AND R_TRIG_1.Q THEN
	IndexData[19]:=IndexData[18];
	IndexData[18]:=IndexData[17];
	IndexData[17]:=IndexData[16];
	IndexData[16]:=IndexData[15];
	IndexData[15]:=IndexData[14];
	IndexData[14]:=IndexData[13];
	IndexData[13]:=IndexData[12];
	IndexData[12]:=IndexData[11];
	IndexData[11]:=IndexData[10];
	IndexData[10]:=IndexData[9];
	IndexData[9]:=IndexData[8];
	IndexData[8]:=IndexData[7];
	IndexData[7]:=IndexData[6];
	IndexData[6]:=IndexData[5];
	IndexData[5]:=IndexData[4];
	IndexData[4]:=IndexData[3];
	IndexData[3]:=IndexData[2];
	IndexData[2]:=IndexData[1];
	IndexData[1]:=IndexData[0];
END_IF;
END_PROGRAM

PROGRAM prIndex
VAR
    R_TRIG_1 : R_TRIG;
    R_TRIG_CT : R_TRIG;
    tDelayTime : TIME;
    TON_1 : TON;
    IndexCanRunStatus : BOOL;
    Autoflow : INT;
    ia : INT;
    ii : INT;
    jj : DINT;
    TON_CT : TON;
END_VAR
VAR_EXTERNAL
    SystemReadyStatus : BOOL;
    HMIPB_RY_Index : BOOL;
    HMISV_Index_DelayTime : DINT;
    YAMAHA_ORG : BOOL;
    LS_S2_UpDownBack : BOOL;
    SOL_S2_UpDown : BOOL;
    LS_S4_UpDownBack : BOOL;
    RY_Index : BOOL;
    ErrorStatus : ARRAY[0..19] OF BOOL;
    AutoStatus : BOOL;
    MachineRunStatus : BOOL;
    IndexData : ARRAY[0..19] OF stIndexData;
    SNR_Index : BOOL;
    SOL_S4_UpDown : BOOL;
    LS_S4_MoveBack : BOOL;
    LS_S6_UpDownBack : BOOL;
    SOL_S6_UpDown : BOOL;
    LS_S6_MoveBack : BOOL;
    LS_S8_UpDownBack : BOOL;
    SOL_S8_UpDown : BOOL;
    LS_S8_MoveOut : BOOL;
    LS_S10_UpDownBack : BOOL;
    SOL_S10_UpDown : BOOL;
    LS_S10_MoveOut : BOOL;
    LS_S11_UpDownBack : BOOL;
    SOL_S11_UpDown : BOOL;
    LS_S13_UpDownBack : BOOL;
    SOL_S13_UpDown : BOOL;
    LS_S15_UpDownBack : BOOL;
    SOL_S15_UpDown : BOOL;
    Error_PB_EStop : BOOL;
    CurrentCycleTime : ARRAY[0..9] OF DINT;
    AverageCycleTime : DINT;
END_VAR
(*************************************************************************
程序名稱:轉盤程式
作者:蔡相偉
版本,日期,版本資訊:
1.0.0	2017/8/8		初始版本
流程
PowerOn=0
Idle=1
轉盤定位回=2
轉盤起動=3
轉盤運轉中=4
轉盤停止=5
轉盤定位出=6
*************************************************************************)
(*PowerOn=0*)
IF NOT(SystemReadyStatus) OR ErrorStatus[0] OR Error_PB_EStop THEN
	AutoFlow:=0;
END_IF;
(*Idle=1*)
IF AutoFlow=0 AND SystemReadyStatus AND NOT(ErrorStatus[0]) AND NOT(Error_PB_EStop) THEN
	AutoFlow:=1;
END_IF;
IF Autoflow=6 AND TON_1.Q THEN
	Autoflow:=1;
END_IF;
(*轉盤定位回=2*)
R_TRIG_1(CLK:= HMIPB_RY_Index AND NOT(AutoStatus));
IF Autoflow=1 AND IndexCanRunStatus AND (R_TRIG_1.Q OR
	(MachineRunStatus AND
	IndexData[1].FinishFlag[1] AND
	IndexData[2].FinishFlag[2] AND
	IndexData[4].FinishFlag[4] AND
	IndexData[5].FinishFlag[5] AND
	IndexData[6].FinishFlag[6] AND
	IndexData[7].FinishFlag[7] AND
	IndexData[8].FinishFlag[8] AND
	IndexData[9].FinishFlag[9] AND
	IndexData[10].FinishFlag[10] AND
	IndexData[11].FinishFlag[11] AND
	IndexData[13].FinishFlag[13] AND
	IndexData[15].FinishFlag[15] AND
	IndexData[16].FinishFlag[16])) THEN
	Autoflow:=2;
END_IF;

(*轉盤起動=3*)
IF Autoflow=2 THEN
	Autoflow:=3;
END_IF;

(*轉盤運轉中=4*)
IF Autoflow=3 AND NOT(SNR_Index) THEN
	Autoflow:=4;
END_IF;

(*轉盤停止=5*)
IF Autoflow=4 AND SNR_Index THEN
	Autoflow:=5;
END_IF;

(*轉盤定位出=6*)
IF Autoflow=5 THEN
	Autoflow:=6;
END_IF;
tDelayTime:=NanoSecToTime(HMISV_Index_DelayTime*100000);
TON_1(IN:= Autoflow=6 ,PT:= tDelayTime);

(******************************************************************)
(*輸出*)
IndexCanRunStatus:=
YAMAHA_ORG AND
(LS_S2_UpDownBack AND NOT(SOL_S2_UpDown)) AND
((LS_S4_UpDownBack AND NOT(SOL_S4_UpDown)) OR NOT(LS_S4_MoveBack)) AND
((LS_S6_UpDownBack AND NOT(SOL_S6_UpDown)) OR NOT(LS_S6_MoveBack)) AND
((LS_S8_UpDownBack AND NOT(SOL_S8_UpDown)) OR NOT(LS_S8_MoveOut)) AND
((LS_S10_UpDownBack AND NOT(SOL_S10_UpDown)) OR NOT(LS_S10_MoveOut)) AND
(LS_S11_UpDownBack AND NOT(SOL_S11_UpDown)) AND
(LS_S13_UpDownBack AND NOT(SOL_S13_UpDown)) AND
(LS_S15_UpDownBack AND NOT(SOL_S15_UpDown));

(*轉盤運轉*)
IF (AutoFlow=3 OR Autoflow=4) AND IndexCanRunStatus THEN
	RY_Index:=TRUE;
	ELSE
	RY_Index:=FALSE;
END_IF;

//*************************************************************
//Cycle Time
//*************************************************************
R_TRIG_CT(CLK:= SNR_Index);
IF R_TRIG_CT.Q AND SystemReadyStatus THEN
	FOR ia:=9 TO 1 BY -1 DO
		CurrentCycleTime[ia]:=CurrentCycleTime[ia-1];
	END_FOR;
	CurrentCycleTime[0]:=LINT_TO_DINT(TimeToNanoSec(TON_CT.ET));
	FOR  ii := 0  TO  9  BY  1  DO
		jj:=jj+ CurrentCycleTime[ii] ;
	END_FOR;
	AverageCycleTime:=jj/10;
	jj:=0;
END_IF;
TON_CT(IN:= MachineRunStatus AND NOT(R_TRIG_CT.Q) ,PT:= t#500s);
END_PROGRAM

PROGRAM prError
VAR
    TON_2 : TON;
    TON_3 : TON;
    ErrorDouble : ARRAY[0..9] of fbErrorDouble;
    ErrorSingle : ARRAY[0..9] of fbErrorSingle;
END_VAR
VAR_EXTERNAL
    SystemReadyStatus : BOOL;
    PB_EStop : BOOL;
    Error_PB_EStop : BOOL;
    SNR_AirSource : BOOL;
    Error_SNR_AirSource : BOOL;
    SNR_S1_Load_Full : BOOL;
    Error_SNR_S1_Load_Full : BOOL;
    SNR_S1_UnLoad_Full : BOOL;
    Error_SNR_S1_UnLoad_Full : BOOL;
    LS_S13_TempHighWarring : BOOL;
    Error_LS_S13_TempHighWarring : BOOL;
    LS_S13_TempLowWarring : BOOL;
    Error_LS_S13_TempLowWarring : BOOL;
    ErrorStatus_MachineStop : BOOL;
    ErrorStatus : ARRAY[0..19] OF BOOL;
    ErrorStatus_TH : ARRAY[0..19] OF BOOL;
    Error_SNR_S1_Load_PanelFeed : BOOL;
    ErrorStatus_S4_Load : BOOL;
    ErrorStatus_S4_UnLoad : BOOL;
    ErrorStatus_S4_Center : BOOL;
    ErrorStatus_MachineNonStop : BOOL;
    Error_SNR_S4_Load_Full : BOOL;
    Error_SNR_S4_UnLoad_Full : BOOL;
    Error_SNR_S6_Full : BOOL;
    Error_SNR_S8_Full : BOOL;
    Error_SNR_S10_Full : BOOL;
    IndexData : ARRAY[0..19] OF stIndexData;
    ErrorStatus_MachineStop_Record : BOOL;
    HMIPB_PB_Reset : BOOL;
    PB_Reset : BOOL;
    ErrorStatus_S1_Load : BOOL;
    ErrorStatus_S1_UnLoad : BOOL;
    ErrorStatus_S8_Fix : BOOL;
    SNR_S1_Door1 : BOOL;
    Error_LS_Door : BOOL;
    SNR_S1_Door2 : BOOL;
    SNR_S1_Door3 : BOOL;
    SNR_S1_Door4 : BOOL;
END_VAR
(*緊急停止*)
IF SystemReadyStatus AND NOT(PB_EStop) THEN
	Error_PB_EStop:=TRUE;
END_IF;
//**********************************************************************************************************************
(*總氣源*)
IF SystemReadyStatus AND NOT(SNR_AirSource) THEN
	Error_SNR_AirSource:=TRUE;
END_IF;
//**********************************************************************************************************************
//第1站出盤無料
TON_2(IN:= (SNR_S1_Load_Full) ,PT:= t#1s);
IF TON_2.Q THEN
	Error_SNR_S1_Load_Full:=TRUE;
ELSE
	Error_SNR_S1_Load_Full:=FALSE;
END_IF;
//**********************************************************************************************************************
//第1站收盤滿料
TON_3(IN:= NOT(SNR_S1_UnLoad_Full) ,PT:= t#1s);
IF TON_3.Q THEN
	Error_SNR_S1_UnLoad_Full:=TRUE;
ELSE
	Error_SNR_S1_UnLoad_Full:=FALSE;
END_IF;
//**********************************************************************************************************************
//第13站溫度過高
IF SystemReadyStatus AND LS_S13_TempHighWarring THEN
	Error_LS_S13_TempHighWarring:=TRUE;
END_IF;
//**********************************************************************************************************************
//第13站溫度過低
IF SystemReadyStatus AND LS_S13_TempLowWarring THEN
	Error_LS_S13_TempLowWarring:=TRUE;
END_IF;
//**********************************************************************************************************************
//門檢
IF SystemReadyStatus AND
	(NOT(SNR_S1_Door1) OR NOT(SNR_S1_Door2) OR NOT(SNR_S1_Door3) OR NOT(SNR_S1_Door4)) THEN
	Error_LS_Door:=TRUE;
END_IF;
//**********************************************************************************************************************
(*機器停機異常*)
ErrorStatus_MachineStop:=
ErrorStatus[0] OR
ErrorStatus[1] OR
ErrorStatus[2] OR
ErrorStatus[3] OR
ErrorStatus[4] OR
ErrorStatus[5] OR
ErrorStatus[6] OR
ErrorStatus[7] OR
ErrorStatus[8] OR
ErrorStatus[9] OR
ErrorStatus[10] OR 
ErrorStatus[11] OR
ErrorStatus[12] OR
ErrorStatus[13] OR
ErrorStatus[14] OR
ErrorStatus[15] OR
ErrorStatus[16] OR
ErrorStatus_TH[1] OR
ErrorStatus_TH[2] OR
ErrorStatus_TH[3] OR
ErrorStatus_TH[4] OR
ErrorStatus_TH[5] OR
ErrorStatus_TH[6] OR
ErrorStatus_TH[7] OR
ErrorStatus_TH[8] OR
ErrorStatus_TH[9] OR
ErrorStatus_TH[10] OR
ErrorStatus_TH[11] OR
ErrorStatus_TH[12] OR
ErrorStatus_TH[13] OR
ErrorStatus_TH[14] OR
ErrorStatus_TH[15] OR
ErrorStatus_TH[16] OR
Error_PB_EStop OR
Error_SNR_AirSource OR
Error_SNR_S1_Load_PanelFeed OR
ErrorStatus_S1_Load OR
ErrorStatus_S1_UnLoad OR
ErrorStatus_S4_Load OR
ErrorStatus_S4_UnLoad OR
ErrorStatus_S4_Center OR
ErrorStatus_S8_Fix OR
Error_LS_S13_TempHighWarring OR
Error_LS_S13_TempLowWarring;
(*機器不停機異常*)
ErrorStatus_MachineNonStop:=
Error_SNR_S1_Load_Full OR
Error_SNR_S1_UnLoad_Full OR
Error_SNR_S4_Load_Full OR
Error_SNR_S4_UnLoad_Full OR
Error_SNR_S6_Full OR
Error_SNR_S8_Full OR
Error_SNR_S10_Full;
(*NG品排除*)
IF IndexData[17].ErrorLog[4]+
	IndexData[17].ErrorLog[5]+
	IndexData[17].ErrorLog[6]+
	IndexData[17].ErrorLog[7]+
	IndexData[17].ErrorLog[8]+
	IndexData[17].ErrorLog[9]+
	IndexData[17].ErrorLog[10]+
	IndexData[17].ErrorLog[11]+
	IndexData[17].ErrorLog[12]+
	IndexData[17].ErrorLog[13]+
	IndexData[17].ErrorLog[14]+
	IndexData[17].ErrorLog[15]+
	IndexData[17].ErrorLog[16]>0
	 THEN
	ErrorStatus_MachineStop_Record:=TRUE;
	ELSE
	ErrorStatus_MachineStop_Record:=FALSE;
END_IF;
//**********************************************************************************************************************
//異常RESET
IF PB_Reset OR HMIPB_PB_Reset THEN
	IndexData[17].ErrorLog[1]:=0;
	IndexData[17].ErrorLog[2]:=0;
	IndexData[17].ErrorLog[3]:=0;
	IndexData[17].ErrorLog[4]:=0;
	IndexData[17].ErrorLog[5]:=0;
	IndexData[17].ErrorLog[6]:=0;
	IndexData[17].ErrorLog[7]:=0;
	IndexData[17].ErrorLog[8]:=0;
	IndexData[17].ErrorLog[9]:=0;
	IndexData[17].ErrorLog[10]:=0;
	IndexData[17].ErrorLog[11]:=0;
	IndexData[17].ErrorLog[12]:=0;
	IndexData[17].ErrorLog[13]:=0;
	IndexData[17].ErrorLog[14]:=0;
	IndexData[17].ErrorLog[15]:=0;
	IndexData[17].ErrorLog[16]:=0;
	Error_PB_EStop:=FALSE;
	Error_SNR_AirSource:=FALSE;
	Error_SNR_S1_Load_PanelFeed:=FALSE;
	Error_LS_S13_TempHighWarring:=FALSE;
	Error_LS_S13_TempLowWarring:=FALSE;
	Error_LS_Door:=FALSE;
END_IF;
END_PROGRAM

PROGRAM prError_S0
VAR
    TON_1 : TON;
END_VAR
VAR_EXTERNAL
    RY_Index : BOOL;
    Error_SNR_Index : BOOL;
    SystemReadyStatus : BOOL;
    Invertor_Ready : BOOL;
    Error_Invertor_Ready : BOOL;
    ErrorStatus : ARRAY[0..19] OF BOOL;
    PB_Reset : BOOL;
    HMIPB_PB_Reset : BOOL;
END_VAR
//**********************************************************************************************************************
//Station0
//**********************************************************************************************************************
(*轉盤微動開關*)
TON_1(IN:= RY_Index ,PT:= t#6s);
IF TON_1.Q THEN
	Error_SNR_Index:=TRUE;
END_IF;

(*變頻器*)
IF SystemReadyStatus AND Invertor_Ready THEN
	Error_Invertor_Ready:=TRUE;
END_IF;

(*異常*)
ErrorStatus[0]:=
Error_SNR_index OR
Error_Invertor_Ready;
//**********************************************************************************************************************
//異常RESET
IF PB_Reset OR HMIPB_PB_Reset THEN
	Error_SNR_index:=FALSE;
	Error_Invertor_Ready:=FALSE;
END_IF;
END_PROGRAM

PROGRAM prError_S1
VAR
    ErrorDouble : ARRAY[0..9] of fbErrorDouble;
    ErrorSingle : ARRAY[0..15] of fbErrorSingle;
END_VAR
VAR_EXTERNAL
    AutoStatus : BOOL;
    PB_Reset : BOOL;
    HMIPB_PB_Reset : BOOL;
    LS_S1_Load_PanelUpDown1Back : BOOL;
    LS_S1_Load_PanelUpDown1Out : BOOL;
    SOL_S1_Load_PanelUpDown1Back : BOOL;
    SOL_S1_Load_PanelUpDown1Out : BOOL;
    Error_LS_S1_Load_PanelUpDown1Back : BOOL;
    Error_LS_S1_Load_PanelUpDown1Out : BOOL;
    LS_S1_Load_PanelUpDown2Back : BOOL;
    LS_S1_Load_PanelUpDown2Out : BOOL;
    SOL_S1_Load_PanelUpDown2Back : BOOL;
    SOL_S1_Load_PanelUpDown2Out : BOOL;
    Error_LS_S1_Load_PanelUpDown2Back : BOOL;
    Error_LS_S1_Load_PanelUpDown2Out : BOOL;
    LS_S1_Load_PanelClip1Back : BOOL;
    LS_S1_Load_PanelClip1Out : BOOL;
    SOL_S1_Load_PanelClip : BOOL;
    Error_LS_S1_Load_PanelClip1Back : BOOL;
    Error_LS_S1_Load_PanelClip1Out : BOOL;
    LS_S1_Load_PanelClip2Back : BOOL;
    LS_S1_Load_PanelClip2Out : BOOL;
    Error_LS_S1_Load_PanelClip2Back : BOOL;
    Error_LS_S1_Load_PanelClip2Out : BOOL;
    LS_S1_Load_FixClipBack : BOOL;
    LS_S1_Load_FixClipOut : BOOL;
    SOL_S1_Load_FixClip : BOOL;
    Error_LS_S1_Load_FixClipBack : BOOL;
    Error_LS_S1_Load_FixClipOut : BOOL;
    LS_S1_Load_AlignmentClipBack : BOOL;
    LS_S1_Load_AlignmentClipOut : BOOL;
    SOL_S1_Load_AlignmentClip : BOOL;
    Error_LS_S1_Load_AlignmentClipBack : BOOL;
    Error_LS_S1_Load_AlignmentClipOut : BOOL;
    LS_S1_Load_ConveyorClip1Back : BOOL;
    LS_S1_Load_ConveyorClip1Out : BOOL;
    SOL_S1_Load_ConveyorClip : BOOL;
    Error_LS_S1_Load_ConveyorClip1Back : BOOL;
    Error_LS_S1_Load_ConveyorClip1Out : BOOL;
    LS_S1_Load_ConveyorClip2Back : BOOL;
    LS_S1_Load_ConveyorClip2Out : BOOL;
    Error_LS_S1_Load_ConveyorClip2Back : BOOL;
    Error_LS_S1_Load_ConveyorClip2Out : BOOL;
    LS_S1_Load_UpDownBack : BOOL;
    LS_S1_Load_UpDownOut : BOOL;
    SOL_S1_Load_UpDown : BOOL;
    Error_LS_S1_Load_UpDownBack : BOOL;
    Error_LS_S1_Load_UpDownOut : BOOL;
    ErrorStatus_S1_Load : BOOL;
    ErrorStatus_S1_FeedPanelLoad : BOOL;
    LS_S1_UnLoad_PanelUpDown1Back : BOOL;
    LS_S1_UnLoad_PanelUpDown1Out : BOOL;
    SOL_S1_UnLoad_PanelUpDown1Back : BOOL;
    SOL_S1_UnLoad_PanelUpDown1Out : BOOL;
    Error_LS_S1_UnLoad_PanelUpDown1Back : BOOL;
    Error_LS_S1_UnLoad_PanelUpDown1Out : BOOL;
    LS_S1_UnLoad_PanelUpDown2Back : BOOL;
    LS_S1_UnLoad_PanelUpDown2Out : BOOL;
    SOL_S1_UnLoad_PanelUpDown2Back : BOOL;
    SOL_S1_UnLoad_PanelUpDown2Out : BOOL;
    Error_LS_S1_UnLoad_PanelUpDown2Out : BOOL;
    Error_LS_S1_UnLoad_PanelUpDown2Back : BOOL;
    LS_S1_UnLoad_PanelClip1Back : BOOL;
    LS_S1_UnLoad_PanelClip1Out : BOOL;
    SOL_S1_UnLoad_PanelClip : BOOL;
    Error_LS_S1_UnLoad_PanelClip1Back : BOOL;
    Error_LS_S1_UnLoad_PanelClip1Out : BOOL;
    LS_S1_UnLoad_PanelClip2Back : BOOL;
    LS_S1_UnLoad_PanelClip2Out : BOOL;
    Error_LS_S1_UnLoad_PanelClip2Back : BOOL;
    Error_LS_S1_UnLoad_PanelClip2Out : BOOL;
    LS_S1_UnLoad_FixClipBack : BOOL;
    LS_S1_UnLoad_FixClipOut : BOOL;
    SOL_S1_UnLoad_FixClip : BOOL;
    Error_LS_S1_UnLoad_FixClipBack : BOOL;
    Error_LS_S1_UnLoad_FixClipOut : BOOL;
    LS_S1_UnLoad_AlignmentClipBack : BOOL;
    LS_S1_UnLoad_AlignmentClipOut : BOOL;
    SOL_S1_UnLoad_AlignmentClip : BOOL;
    Error_LS_S1_UnLoad_AlignmentClipBack : BOOL;
    Error_LS_S1_UnLoad_AlignmentClipOut : BOOL;
    LS_S1_UnLoad_ConveyorClip1Back : BOOL;
    LS_S1_UnLoad_ConveyorClip1Out : BOOL;
    SOL_S1_UnLoad_ConveyorClip : BOOL;
    Error_LS_S1_UnLoad_ConveyorClip1Back : BOOL;
    Error_LS_S1_UnLoad_ConveyorClip1Out : BOOL;
    LS_S1_UnLoad_ConveyorClip2Back : BOOL;
    LS_S1_UnLoad_ConveyorClip2Out : BOOL;
    Error_LS_S1_UnLoad_ConveyorClip2Back : BOOL;
    Error_LS_S1_UnLoad_ConveyorClip2Out : BOOL;
    LS_S1_UnLoad_UpDownBack : BOOL;
    LS_S1_UnLoad_UpDownOut : BOOL;
    SOL_S1_UnLoad_UpDown : BOOL;
    Error_LS_S1_UnLoad_UpDownBack : BOOL;
    Error_LS_S1_UnLoad_UpDownOut : BOOL;
    ErrorStatus_S1_UnLoad : BOOL;
    ErrorStatus_S1_FeedPanelUnLoad : BOOL;
    ErrorStatus_TH : ARRAY[0..19] OF BOOL;
    ErrorStatus : ARRAY[0..19] OF BOOL;
    YAMAHA_S_State_Alarm : BOOL;
    YAMAHA_S_State_Warring : BOOL;
    YAMAHA_Error_SOL_Clip : BOOL;
    Error_SNR_S1_Load_PanelFeed : BOOL;
END_VAR
//**********************************************************************************************************************
(*Station1*)
//**********************************************************************************************************************
//LOAD
ErrorDouble[0](
	bAutoStatus:=AutoStatus,
	bResetPB:=PB_Reset OR HMIPB_PB_Reset,
	bBackLS:=LS_S1_Load_PanelUpDown1Back,
	bOutLS:=LS_S1_Load_PanelUpDown1Out,
	bBackSOL:=SOL_S1_Load_PanelUpDown1Back,
	bOutSOL:=SOL_S1_Load_PanelUpDown1Out,
	bErrorStatus_Back=>Error_LS_S1_Load_PanelUpDown1Back,
	bErrorStatus_Out=>Error_LS_S1_Load_PanelUpDown1Out);

ErrorDouble[1](
	bAutoStatus:=AutoStatus,
	bResetPB:=PB_Reset OR HMIPB_PB_Reset,
	bBackLS:=LS_S1_Load_PanelUpDown2Back,
	bOutLS:=LS_S1_Load_PanelUpDown2Out,
	bBackSOL:=SOL_S1_Load_PanelUpDown2Back,
	bOutSOL:=SOL_S1_Load_PanelUpDown2Out,
	bErrorStatus_Back=>Error_LS_S1_Load_PanelUpDown2Back,
	bErrorStatus_Out=>Error_LS_S1_Load_PanelUpDown2Out);

ErrorSingle[0](
	bAutoStatus:=AutoStatus,
	bResetPB:=PB_Reset OR HMIPB_PB_Reset,
	bBackLS:=LS_S1_Load_PanelClip1Back,
	bOutLS:=LS_S1_Load_PanelClip1Out,
	bSOL:=SOL_S1_Load_PanelClip,
	bErrorStatus_Back=>Error_LS_S1_Load_PanelClip1Back,
	bErrorStatus_Out=>Error_LS_S1_Load_PanelClip1Out);

ErrorSingle[1](
	bAutoStatus:=AutoStatus,
	bResetPB:=PB_Reset OR HMIPB_PB_Reset,
	bBackLS:=LS_S1_Load_PanelClip2Back,
	bOutLS:=LS_S1_Load_PanelClip2Out,
	bSOL:=SOL_S1_Load_PanelClip,
	bErrorStatus_Back=>Error_LS_S1_Load_PanelClip2Back,
	bErrorStatus_Out=>Error_LS_S1_Load_PanelClip2Out);

//Load取料位
ErrorSingle[2](
	bAutoStatus:=AutoStatus,
	bResetPB:=PB_Reset OR HMIPB_PB_Reset,
	bBackLS:=LS_S1_Load_FixClipBack,
	bOutLS:=LS_S1_Load_FixClipOut,
	bSOL:=SOL_S1_Load_FixClip,
	bErrorStatus_Back=>Error_LS_S1_Load_FixClipBack,
	bErrorStatus_Out=>Error_LS_S1_Load_FixClipOut);

ErrorSingle[3](
	bAutoStatus:=AutoStatus,
	bResetPB:=PB_Reset OR HMIPB_PB_Reset,
	bBackLS:=LS_S1_Load_AlignmentClipBack,
	bOutLS:=LS_S1_Load_AlignmentClipOut,
	bSOL:=SOL_S1_Load_AlignmentClip,
	bErrorStatus_Back=>Error_LS_S1_Load_AlignmentClipBack,
	bErrorStatus_Out=>Error_LS_S1_Load_AlignmentClipOut);

ErrorSingle[4](
	bAutoStatus:=AutoStatus,
	bResetPB:=PB_Reset OR HMIPB_PB_Reset,
	bBackLS:=LS_S1_Load_ConveyorClip1Back,
	bOutLS:=LS_S1_Load_ConveyorClip1Out,
	bSOL:=SOL_S1_Load_ConveyorClip,
	bErrorStatus_Back=>Error_LS_S1_Load_ConveyorClip1Back,
	bErrorStatus_Out=>Error_LS_S1_Load_ConveyorClip1Out);

ErrorSingle[5](
	bAutoStatus:=AutoStatus,
	bResetPB:=PB_Reset OR HMIPB_PB_Reset,
	bBackLS:=LS_S1_Load_ConveyorClip2Back,
	bOutLS:=LS_S1_Load_ConveyorClip2Out,
	bSOL:=SOL_S1_Load_ConveyorClip,
	bErrorStatus_Back=>Error_LS_S1_Load_ConveyorClip2Back,
	bErrorStatus_Out=>Error_LS_S1_Load_ConveyorClip2Out);

ErrorSingle[6](
	bAutoStatus:=AutoStatus,
	bResetPB:=PB_Reset OR HMIPB_PB_Reset,
	bBackLS:=LS_S1_Load_UpDownBack,
	bOutLS:=LS_S1_Load_UpDownOut,
	bSOL:=SOL_S1_Load_UpDown,
	bErrorStatus_Back=>Error_LS_S1_Load_UpDownBack,
	bErrorStatus_Out=>Error_LS_S1_Load_UpDownOut);

//異常
ErrorStatus_S1_Load:=
Error_LS_S1_Load_PanelUpDown1Back OR
Error_LS_S1_Load_PanelUpDown1Out OR
Error_LS_S1_Load_PanelUpDown2Back OR
Error_LS_S1_Load_PanelUpDown2Out OR
Error_LS_S1_Load_PanelClip1Back OR
Error_LS_S1_Load_PanelClip1Out OR
Error_LS_S1_Load_PanelClip2Back OR
Error_LS_S1_Load_PanelClip2Out;

ErrorStatus_S1_FeedPanelLoad:=
Error_LS_S1_Load_FixClipBack OR
Error_LS_S1_Load_FixClipOut OR
Error_LS_S1_Load_AlignmentClipBack OR
Error_LS_S1_Load_AlignmentClipOut OR
Error_LS_S1_Load_ConveyorClip1Back OR
Error_LS_S1_Load_ConveyorClip1Out OR
Error_LS_S1_Load_ConveyorClip2Back OR
Error_LS_S1_Load_ConveyorClip2Out OR
Error_LS_S1_Load_UpDownBack OR
Error_LS_S1_Load_UpDownOut;

//UNLOAD
ErrorDouble[2](
	bAutoStatus:=AutoStatus,
	bResetPB:=PB_Reset OR HMIPB_PB_Reset,
	bBackLS:=LS_S1_UnLoad_PanelUpDown1Back,
	bOutLS:=LS_S1_UnLoad_PanelUpDown1Out,
	bBackSOL:=SOL_S1_UnLoad_PanelUpDown1Back,
	bOutSOL:=SOL_S1_UnLoad_PanelUpDown1Out,
	bErrorStatus_Back=>Error_LS_S1_UnLoad_PanelUpDown1Back,
	bErrorStatus_Out=>Error_LS_S1_UnLoad_PanelUpDown1Out);

ErrorDouble[3](
	bAutoStatus:=AutoStatus,
	bResetPB:=PB_Reset OR HMIPB_PB_Reset,
	bBackLS:=LS_S1_UnLoad_PanelUpDown2Back,
	bOutLS:=LS_S1_UnLoad_PanelUpDown2Out,
	bBackSOL:=SOL_S1_UnLoad_PanelUpDown2Back,
	bOutSOL:=SOL_S1_UnLoad_PanelUpDown2Out,
	bErrorStatus_Back=>Error_LS_S1_UnLoad_PanelUpDown2Back,
	bErrorStatus_Out=>Error_LS_S1_UnLoad_PanelUpDown2Out);

ErrorSingle[7](
	bAutoStatus:=AutoStatus,
	bResetPB:=PB_Reset OR HMIPB_PB_Reset,
	bBackLS:=LS_S1_UnLoad_PanelClip1Back,
	bOutLS:=LS_S1_UnLoad_PanelClip1Out,
	bSOL:=SOL_S1_UnLoad_PanelClip,
	bErrorStatus_Back=>Error_LS_S1_UnLoad_PanelClip1Back,
	bErrorStatus_Out=>Error_LS_S1_UnLoad_PanelClip1Out);

ErrorSingle[8](
	bAutoStatus:=AutoStatus,
	bResetPB:=PB_Reset OR HMIPB_PB_Reset,
	bBackLS:=LS_S1_UnLoad_PanelClip2Back,
	bOutLS:=LS_S1_UnLoad_PanelClip2Out,
	bSOL:=SOL_S1_UnLoad_PanelClip,
	bErrorStatus_Back=>Error_LS_S1_UnLoad_PanelClip2Back,
	bErrorStatus_Out=>Error_LS_S1_UnLoad_PanelClip2Out);

//UNLoad放料位
ErrorSingle[9](
	bAutoStatus:=AutoStatus,
	bResetPB:=PB_Reset OR HMIPB_PB_Reset,
	bBackLS:=LS_S1_UnLoad_FixClipBack,
	bOutLS:=LS_S1_UnLoad_FixClipOut,
	bSOL:=SOL_S1_UnLoad_FixClip,
	bErrorStatus_Back=>Error_LS_S1_UnLoad_FixClipBack,
	bErrorStatus_Out=>Error_LS_S1_UnLoad_FixClipOut);

ErrorSingle[10](
	bAutoStatus:=AutoStatus,
	bResetPB:=PB_Reset OR HMIPB_PB_Reset,
	bBackLS:=LS_S1_UnLoad_AlignmentClipBack,
	bOutLS:=LS_S1_UnLoad_AlignmentClipOut,
	bSOL:=SOL_S1_UnLoad_AlignmentClip,
	bErrorStatus_Back=>Error_LS_S1_UnLoad_AlignmentClipBack,
	bErrorStatus_Out=>Error_LS_S1_UnLoad_AlignmentClipOut);

ErrorSingle[11](
	bAutoStatus:=AutoStatus,
	bResetPB:=PB_Reset OR HMIPB_PB_Reset,
	bBackLS:=LS_S1_UnLoad_ConveyorClip1Back,
	bOutLS:=LS_S1_UnLoad_ConveyorClip1Out,
	bSOL:=SOL_S1_UnLoad_ConveyorClip,
	bErrorStatus_Back=>Error_LS_S1_UnLoad_ConveyorClip1Back,
	bErrorStatus_Out=>Error_LS_S1_UnLoad_ConveyorClip1Out);

ErrorSingle[12](
	bAutoStatus:=AutoStatus,
	bResetPB:=PB_Reset OR HMIPB_PB_Reset,
	bBackLS:=LS_S1_UnLoad_ConveyorClip2Back,
	bOutLS:=LS_S1_UnLoad_ConveyorClip2Out,
	bSOL:=SOL_S1_UnLoad_ConveyorClip,
	bErrorStatus_Back=>Error_LS_S1_UnLoad_ConveyorClip2Back,
	bErrorStatus_Out=>Error_LS_S1_UnLoad_ConveyorClip2Out);

ErrorSingle[13](
	bAutoStatus:=AutoStatus,
	bResetPB:=PB_Reset OR HMIPB_PB_Reset,
	bBackLS:=LS_S1_UnLoad_UpDownBack,
	bOutLS:=LS_S1_UnLoad_UpDownOut,
	bSOL:=SOL_S1_UnLoad_UpDown,
	bErrorStatus_Back=>Error_LS_S1_UnLoad_UpDownBack,
	bErrorStatus_Out=>Error_LS_S1_UnLoad_UpDownOut);
//異常
ErrorStatus_S1_UnLoad:=
Error_LS_S1_UnLoad_PanelUpDown1Back OR
Error_LS_S1_UnLoad_PanelUpDown1Out OR
Error_LS_S1_UnLoad_PanelUpDown2Back OR
Error_LS_S1_UnLoad_PanelUpDown2Out OR
Error_LS_S1_UnLoad_PanelClip1Back OR
Error_LS_S1_UnLoad_PanelClip1Out OR
Error_LS_S1_UnLoad_PanelClip2Back OR
Error_LS_S1_UnLoad_PanelClip2Out;

ErrorStatus_S1_FeedPanelUnLoad:=
Error_LS_S1_UnLoad_FixClipBack OR
Error_LS_S1_UnLoad_FixClipOut OR
Error_LS_S1_UnLoad_AlignmentClipBack OR
Error_LS_S1_UnLoad_AlignmentClipOut OR
Error_LS_S1_UnLoad_ConveyorClip1Back OR
Error_LS_S1_UnLoad_ConveyorClip1Out OR
Error_LS_S1_UnLoad_ConveyorClip2Back OR
Error_LS_S1_UnLoad_ConveyorClip2Out OR
Error_LS_S1_UnLoad_UpDownBack OR
Error_LS_S1_UnLoad_UpDownOut;

ErrorStatus_TH[1]:=
ErrorStatus_S1_FeedPanelLoad OR
ErrorStatus_S1_FeedPanelUnLoad;

ErrorStatus[1]:=
YAMAHA_S_State_Alarm OR
YAMAHA_S_State_Warring OR
YAMAHA_Error_SOL_Clip OR
ErrorStatus_TH[1];
//**********************************************************************************************************************
//異常RESET
IF PB_Reset OR HMIPB_PB_Reset THEN
	Error_SNR_S1_Load_PanelFeed:=FALSE;
END_IF;
END_PROGRAM

PROGRAM prError_S2
VAR
    ErrorSingle : ARRAY[0..1] of fbErrorSingle;
END_VAR
VAR_EXTERNAL
    AutoStatus : BOOL;
    PB_Reset : BOOL;
    HMIPB_PB_Reset : BOOL;
    LS_S2_UpDownBack : BOOL;
    LS_S2_UpDownOut : BOOL;
    SOL_S2_UpDown : BOOL;
    Error_LS_S2_UpDownBack : BOOL;
    Error_LS_S2_UpDownOut : BOOL;
    ErrorStatus : ARRAY[0..19] OF BOOL;
END_VAR
//**********************************************************************************************************************
(*Station2*)
//**********************************************************************************************************************
ErrorSingle[0](
	bAutoStatus:=AutoStatus,
	bResetPB:=PB_Reset OR HMIPB_PB_Reset,
	bBackLS:=LS_S2_UpDownBack,
	bOutLS:=LS_S2_UpDownOut,
	bSOL:=SOL_S2_UpDown,
	bErrorStatus_Back=>Error_LS_S2_UpDownBack,
	bErrorStatus_Out=>Error_LS_S2_UpDownOut);

ErrorStatus[2]:=
Error_LS_S2_UpDownBack OR
Error_LS_S2_UpDownOut;
END_PROGRAM

PROGRAM prError_S4
VAR
    ErrorDouble : ARRAY[0..9] of fbErrorDouble;
    ErrorSingle : ARRAY[0..9] of fbErrorSingle;
END_VAR
VAR_EXTERNAL
    AutoStatus : BOOL;
    PB_Reset : BOOL;
    HMIPB_PB_Reset : BOOL;
    LS_S4_MoveBack : BOOL;
    LS_S4_MoveOut : BOOL;
    SOL_S4_MoveBack : BOOL;
    SOL_S4_MoveOut : BOOL;
    Error_LS_S4_MoveBack : BOOL;
    Error_LS_S4_MoveOut : BOOL;
    LS_S4_UpDownBack : BOOL;
    LS_S4_UpDownOut : BOOL;
    SOL_S4_UpDown : BOOL;
    Error_LS_S4_UpDownBack : BOOL;
    Error_LS_S4_UpDownOut : BOOL;
    LS_S4_ClipBack : BOOL;
    LS_S4_ClipOut : BOOL;
    SOL_S4_Clip : BOOL;
    Error_LS_S4_ClipBack : BOOL;
    Error_LS_S4_ClipOut : BOOL;
    LS_S4_THMoveBack : BOOL;
    LS_S4_THMoveOut : BOOL;
    SOL_S4_THMoveBack : BOOL;
    SOL_S4_THMoveOut : BOOL;
    Error_LS_S4_THMoveBack : BOOL;
    Error_LS_S4_THMoveOut : BOOL;
    LS_S4_Load_PanelUpDown1Back : BOOL;
    LS_S4_Load_PanelUpDown1Out : BOOL;
    SOL_S4_Load_PanelUpDown1Back : BOOL;
    SOL_S4_Load_PanelUpDown1Out : BOOL;
    Error_LS_S4_Load_PanelUpDown1Back : BOOL;
    Error_LS_S4_Load_PanelUpDown1Out : BOOL;
    LS_S4_Load_PanelUpDown2Back : BOOL;
    LS_S4_Load_PanelUpDown2Out : BOOL;
    SOL_S4_Load_PanelUpDown2Back : BOOL;
    SOL_S4_Load_PanelUpDown2Out : BOOL;
    Error_LS_S4_Load_PanelUpDown2Back : BOOL;
    Error_LS_S4_Load_PanelUpDown2Out : BOOL;
    LS_S4_Load_PanelClip1Back : BOOL;
    LS_S4_Load_PanelClip1Out : BOOL;
    SOL_S4_Load_PanelClip : BOOL;
    Error_LS_S4_Load_PanelClip1Back : BOOL;
    Error_LS_S4_Load_PanelClip1Out : BOOL;
    LS_S4_Load_PanelClip2Back : BOOL;
    LS_S4_Load_PanelClip2Out : BOOL;
    Error_LS_S4_Load_PanelClip2Back : BOOL;
    Error_LS_S4_Load_PanelClip2Out : BOOL;
    LS_S4_UnLoad_PanelUpDown1Back : BOOL;
    LS_S4_UnLoad_PanelUpDown1Out : BOOL;
    SOL_S4_UnLoad_PanelUpDown1Back : BOOL;
    SOL_S4_UnLoad_PanelUpDown1Out : BOOL;
    Error_LS_S4_UnLoad_PanelUpDown1Back : BOOL;
    Error_LS_S4_UnLoad_PanelUpDown1Out : BOOL;
    LS_S4_UnLoad_PanelUpDown2Back : BOOL;
    LS_S4_UnLoad_PanelUpDown2Out : BOOL;
    SOL_S4_UnLoad_PanelUpDown2Back : BOOL;
    SOL_S4_UnLoad_PanelUpDown2Out : BOOL;
    Error_LS_S4_UnLoad_PanelUpDown2Back : BOOL;
    Error_LS_S4_UnLoad_PanelUpDown2Out : BOOL;
    LS_S4_UnLoad_PanelClip1Back : BOOL;
    LS_S4_UnLoad_PanelClip1Out : BOOL;
    SOL_S4_UnLoad_PanelClip : BOOL;
    Error_LS_S4_UnLoad_PanelClip1Back : BOOL;
    Error_LS_S4_UnLoad_PanelClip1Out : BOOL;
    LS_S4_UnLoad_PanelClip2Back : BOOL;
    LS_S4_UnLoad_PanelClip2Out : BOOL;
    Error_LS_S4_UnLoad_PanelClip2Back : BOOL;
    Error_LS_S4_UnLoad_PanelClip2Out : BOOL;
    LS_S4_Center_ClipBack : BOOL;
    LS_S4_Center_ClipOut : BOOL;
    SOL_S4_Center_Clip : BOOL;
    Error_LS_S4_Center_ClipBack : BOOL;
    Error_LS_S4_Center_ClipOut : BOOL;
    LS_S4_Center_UpDownBack : BOOL;
    LS_S4_Center_UpDownOut : BOOL;
    Error_LS_S4_Center_UpDownBack : BOOL;
    Error_LS_S4_Center_UpDownOut : BOOL;
    ErrorStatus : ARRAY[0..19] OF BOOL;
    ErrorStatus_TH : ARRAY[0..19] OF BOOL;
    ErrorStatus_S4_Load : BOOL;
    ErrorStatus_S4_UnLoad : BOOL;
    ErrorStatus_S4_Center : BOOL;
END_VAR
//**********************************************************************************************************************
(*Station4*)
//**********************************************************************************************************************
ErrorDouble[0](
	bAutoStatus:=AutoStatus,
	bResetPB:=PB_Reset OR HMIPB_PB_Reset,
	bBackLS:=LS_S4_MoveBack,
	bOutLS:=LS_S4_MoveOut,
	bBackSOL:=SOL_S4_MoveBack,
	bOutSOL:=SOL_S4_MoveOut,
	bErrorStatus_Back=>Error_LS_S4_MoveBack,
	bErrorStatus_Out=>Error_LS_S4_MoveOut);

ErrorSingle[0](
	bAutoStatus:=AutoStatus,
	bResetPB:=PB_Reset OR HMIPB_PB_Reset,
	bBackLS:=LS_S4_UpDownBack,
	bOutLS:=LS_S4_UpDownOut,
	bSOL:=SOL_S4_UpDown,
	bErrorStatus_Back=>Error_LS_S4_UpDownBack,
	bErrorStatus_Out=>Error_LS_S4_UpDownOut);

ErrorSingle[1](
	bAutoStatus:=AutoStatus,
	bResetPB:=PB_Reset OR HMIPB_PB_Reset,
	bBackLS:=LS_S4_ClipBack,
	bOutLS:=LS_S4_ClipOut,
	bSOL:=SOL_S4_Clip,
	bErrorStatus_Back=>Error_LS_S4_ClipBack,
	bErrorStatus_Out=>Error_LS_S4_ClipOut);

ErrorDouble[1](
	bAutoStatus:=AutoStatus,
	bResetPB:=PB_Reset OR HMIPB_PB_Reset,
	bBackLS:=LS_S4_THMoveBack,
	bOutLS:=LS_S4_THMoveOut,
	bBackSOL:=SOL_S4_THMoveBack,
	bOutSOL:=SOL_S4_THMoveOut,
	bErrorStatus_Back=>Error_LS_S4_THMoveBack,
	bErrorStatus_Out=>Error_LS_S4_THMoveOut);

ErrorDouble[2](
	bAutoStatus:=AutoStatus,
	bResetPB:=PB_Reset OR HMIPB_PB_Reset,
	bBackLS:=LS_S4_Load_PanelUpDown1Back,
	bOutLS:=LS_S4_Load_PanelUpDown1Out,
	bBackSOL:=SOL_S4_Load_PanelUpDown1Back,
	bOutSOL:=SOL_S4_Load_PanelUpDown1Out,
	bErrorStatus_Back=>Error_LS_S4_Load_PanelUpDown1Back,
	bErrorStatus_Out=>Error_LS_S4_Load_PanelUpDown1Out);

ErrorDouble[3](
	bAutoStatus:=AutoStatus,
	bResetPB:=PB_Reset OR HMIPB_PB_Reset,
	bBackLS:=LS_S4_Load_PanelUpDown2Back,
	bOutLS:=LS_S4_Load_PanelUpDown2Out,
	bBackSOL:=SOL_S4_Load_PanelUpDown2Back,
	bOutSOL:=SOL_S4_Load_PanelUpDown2Out,
	bErrorStatus_Back=>Error_LS_S4_Load_PanelUpDown2Back,
	bErrorStatus_Out=>Error_LS_S4_Load_PanelUpDown2Out);

ErrorSingle[2](
	bAutoStatus:=AutoStatus,
	bResetPB:=PB_Reset OR HMIPB_PB_Reset,
	bBackLS:=LS_S4_Load_PanelClip1Back,
	bOutLS:=LS_S4_Load_PanelClip1Out,
	bSOL:=SOL_S4_Load_PanelClip,
	bErrorStatus_Back=>Error_LS_S4_Load_PanelClip1Back,
	bErrorStatus_Out=>Error_LS_S4_Load_PanelClip1Out);

ErrorSingle[3](
	bAutoStatus:=AutoStatus,
	bResetPB:=PB_Reset OR HMIPB_PB_Reset,
	bBackLS:=LS_S4_Load_PanelClip2Back,
	bOutLS:=LS_S4_Load_PanelClip2Out,
	bSOL:=SOL_S4_Load_PanelClip,
	bErrorStatus_Back=>Error_LS_S4_Load_PanelClip2Back,
	bErrorStatus_Out=>Error_LS_S4_Load_PanelClip2Out);

ErrorDouble[4](
	bAutoStatus:=AutoStatus,
	bResetPB:=PB_Reset OR HMIPB_PB_Reset,
	bBackLS:=LS_S4_UnLoad_PanelUpDown1Back,
	bOutLS:=LS_S4_UnLoad_PanelUpDown1Out,
	bBackSOL:=SOL_S4_UnLoad_PanelUpDown1Back,
	bOutSOL:=SOL_S4_UnLoad_PanelUpDown1Out,
	bErrorStatus_Back=>Error_LS_S4_UnLoad_PanelUpDown1Back,
	bErrorStatus_Out=>Error_LS_S4_UnLoad_PanelUpDown1Out);

ErrorDouble[5](
	bAutoStatus:=AutoStatus,
	bResetPB:=PB_Reset OR HMIPB_PB_Reset,
	bBackLS:=LS_S4_UnLoad_PanelUpDown2Back,
	bOutLS:=LS_S4_UnLoad_PanelUpDown2Out,
	bBackSOL:=SOL_S4_UnLoad_PanelUpDown2Back,
	bOutSOL:=SOL_S4_UnLoad_PanelUpDown2Out,
	bErrorStatus_Back=>Error_LS_S4_UnLoad_PanelUpDown2Back,
	bErrorStatus_Out=>Error_LS_S4_UnLoad_PanelUpDown2Out);

ErrorSingle[4](
	bAutoStatus:=AutoStatus,
	bResetPB:=PB_Reset OR HMIPB_PB_Reset,
	bBackLS:=LS_S4_UnLoad_PanelClip1Back,
	bOutLS:=LS_S4_UnLoad_PanelClip1Out,
	bSOL:=SOL_S4_UnLoad_PanelClip,
	bErrorStatus_Back=>Error_LS_S4_UnLoad_PanelClip1Back,
	bErrorStatus_Out=>Error_LS_S4_UnLoad_PanelClip1Out);

ErrorSingle[5](
	bAutoStatus:=AutoStatus,
	bResetPB:=PB_Reset OR HMIPB_PB_Reset,
	bBackLS:=LS_S4_UnLoad_PanelClip2Back,
	bOutLS:=LS_S4_UnLoad_PanelClip2Out,
	bSOL:=SOL_S4_UnLoad_PanelClip,
	bErrorStatus_Back=>Error_LS_S4_UnLoad_PanelClip2Back,
	bErrorStatus_Out=>Error_LS_S4_UnLoad_PanelClip2Out);

ErrorSingle[6](
	bAutoStatus:=AutoStatus,
	bResetPB:=PB_Reset OR HMIPB_PB_Reset,
	bBackLS:=LS_S4_Center_ClipBack,
	bOutLS:=LS_S4_Center_ClipOut,
	bSOL:=SOL_S4_Center_Clip,
	bErrorStatus_Back=>Error_LS_S4_Center_ClipBack,
	bErrorStatus_Out=>Error_LS_S4_Center_ClipOut);

ErrorSingle[7](
	bAutoStatus:=AutoStatus,
	bResetPB:=PB_Reset OR HMIPB_PB_Reset,
	bBackLS:=LS_S4_Center_UpDownBack,
	bOutLS:=LS_S4_Center_UpDownOut,
	bSOL:=SOL_S4_Center_Clip,
	bErrorStatus_Back=>Error_LS_S4_Center_UpDownBack,
	bErrorStatus_Out=>Error_LS_S4_Center_UpDownOut);

//異常
ErrorStatus[4]:=
Error_LS_S4_MoveBack OR
Error_LS_S4_MoveBack OR
Error_LS_S4_UpDownBack OR
Error_LS_S4_UpDownOut OR
Error_LS_S4_ClipBack OR
Error_LS_S4_ClipOut;

ErrorStatus_TH[4]:=
Error_LS_S4_THMoveBack OR
Error_LS_S4_THMoveBack;

ErrorStatus_S4_Load:=
Error_LS_S4_Load_PanelUpDown1Back OR
Error_LS_S4_Load_PanelUpDown1Out OR
Error_LS_S4_Load_PanelUpDown2Back OR
Error_LS_S4_Load_PanelUpDown2Out OR
Error_LS_S4_Load_PanelClip1Back OR
Error_LS_S4_Load_PanelClip1Out OR
Error_LS_S4_Load_PanelClip2Back OR
Error_LS_S4_Load_PanelClip2Out;

ErrorStatus_S4_UnLoad:=
Error_LS_S4_UnLoad_PanelUpDown1Back OR
Error_LS_S4_UnLoad_PanelUpDown1Out OR
Error_LS_S4_UnLoad_PanelUpDown2Back OR
Error_LS_S4_UnLoad_PanelUpDown2Out OR
Error_LS_S4_UnLoad_PanelClip1Back OR
Error_LS_S4_UnLoad_PanelClip1Out OR
Error_LS_S4_UnLoad_PanelClip2Back OR
Error_LS_S4_UnLoad_PanelClip2Out;

ErrorStatus_S4_Center:=
Error_LS_S4_Center_UpDownBack OR
Error_LS_S4_Center_UpDownOut OR
Error_LS_S4_Center_ClipBack OR
Error_LS_S4_Center_ClipOut;
END_PROGRAM

PROGRAM prError_S6
VAR
    ErrorDouble : ARRAY[0..9] of fbErrorDouble;
    ErrorSingle : ARRAY[0..9] of fbErrorSingle;
    TON_1 : TON;
END_VAR
VAR_EXTERNAL
    AutoStatus : BOOL;
    PB_Reset : BOOL;
    HMIPB_PB_Reset : BOOL;
    LS_S6_MoveBack : BOOL;
    LS_S6_MoveOut : BOOL;
    SOL_S6_MoveBack : BOOL;
    SOL_S6_MoveOut : BOOL;
    Error_LS_S6_MoveBack : BOOL;
    Error_LS_S6_MoveOut : BOOL;
    LS_S6_UpDownBack : BOOL;
    LS_S6_UpDownOut : BOOL;
    SOL_S6_UpDown : BOOL;
    Error_LS_S6_UpDownBack : BOOL;
    Error_LS_S6_UpDownOut : BOOL;
    SOL_S6_Vacuum : BOOL;
    SNR_S6_Vacuum : BOOL;
    Error_SNR_S6_Vacuum : BOOL;
    ErrorStatus : ARRAY[0..19] OF BOOL;
    ErrorStatus_TH : ARRAY[0..19] OF BOOL;
    LS_S6_THBack : BOOL;
    LS_S6_THOut : BOOL;
    SOL_S6_TH : BOOL;
    Error_LS_S6_THBack : BOOL;
    Error_LS_S6_THOut : BOOL;
END_VAR
//**********************************************************************************************************************
(*Station6*)
//**********************************************************************************************************************
ErrorDouble[0](
	bAutoStatus:=AutoStatus,
	bResetPB:=PB_Reset OR HMIPB_PB_Reset,
	bBackLS:=LS_S6_MoveBack,
	bOutLS:=LS_S6_MoveOut,
	bBackSOL:=SOL_S6_MoveBack,
	bOutSOL:=SOL_S6_MoveOut,
	bErrorStatus_Back=>Error_LS_S6_MoveBack,
	bErrorStatus_Out=>Error_LS_S6_MoveOut);

ErrorSingle[0](
	bAutoStatus:=AutoStatus,
	bResetPB:=PB_Reset OR HMIPB_PB_Reset,
	bBackLS:=LS_S6_UpDownBack,
	bOutLS:=LS_S6_UpDownOut,
	bSOL:=SOL_S6_UpDown,
	bErrorStatus_Back=>Error_LS_S6_UpDownBack,
	bErrorStatus_Out=>Error_LS_S6_UpDownOut);

ErrorSingle[1](
	bAutoStatus:=AutoStatus,
	bResetPB:=PB_Reset OR HMIPB_PB_Reset,
	bBackLS:=LS_S6_THBack,
	bOutLS:=LS_S6_THOut,
	bSOL:=SOL_S6_TH,
	bErrorStatus_Back=>Error_LS_S6_THBack,
	bErrorStatus_Out=>Error_LS_S6_THOut);

TON_1(IN:= SOL_S6_Vacuum AND NOT(SNR_S6_Vacuum) ,PT:= t#2s);
IF TON_1.Q THEN
	Error_SNR_S6_Vacuum:=TRUE;
END_IF;

//異常
ErrorStatus[6]:=
Error_LS_S6_MoveBack OR
Error_LS_S6_MoveBack OR
Error_LS_S6_UpDownBack OR
Error_LS_S6_UpDownOut OR
Error_SNR_S6_Vacuum;

ErrorStatus_TH[6]:=
Error_LS_S6_THBack OR
Error_LS_S6_THOut;
END_PROGRAM

PROGRAM prError_S8
VAR
    ErrorDouble : ARRAY[0..9] of fbErrorDouble;
    ErrorSingle : ARRAY[0..9] of fbErrorSingle;
    TON_1 : TON;
    TON_2 : TON;
END_VAR
VAR_EXTERNAL
    AutoStatus : BOOL;
    PB_Reset : BOOL;
    HMIPB_PB_Reset : BOOL;
    LS_S8_MoveBack : BOOL;
    LS_S8_MoveOut : BOOL;
    SOL_S8_MoveBack : BOOL;
    SOL_S8_MoveOut : BOOL;
    Error_LS_S8_MoveBack : BOOL;
    Error_LS_S8_MoveOut : BOOL;
    LS_S8_UpDownBack : BOOL;
    LS_S8_UpDownOut : BOOL;
    SOL_S8_UpDown : BOOL;
    Error_LS_S8_UpDownBack : BOOL;
    Error_LS_S8_UpDownOut : BOOL;
    ErrorStatus : ARRAY[0..19] OF BOOL;
    ErrorStatus_TH : ARRAY[0..19] OF BOOL;
    LS_S8_THBack : BOOL;
    LS_S8_THOut : BOOL;
    SOL_S8_TH : BOOL;
    Error_LS_S8_THBack : BOOL;
    Error_LS_S8_THOut : BOOL;
    SOL_S8_VacuumF : BOOL;
    SNR_S8_VacuumF : BOOL;
    Error_SNR_S8_VacuumF : BOOL;
    SOL_S8_VacuumR : BOOL;
    SNR_S8_VacuumR : BOOL;
    Error_SNR_S8_VacuumR : BOOL;
    ErrorStatus_S8_Fix : BOOL;
    SystemReadyStatus : BOOL;
    PB_EStop : BOOL;
    Error_PB_EStop : BOOL;
    OMRON_FQ2_Error : BOOL;
    Error_OMRON_FQ2_Error : BOOL;
    LS_S8_FixBack : BOOL;
    LS_S8_FixOut : BOOL;
    SOL_S8_Fix : BOOL;
    Error_LS_S8_FixBack : BOOL;
    Error_LS_S8_FixOut : BOOL;
    LS_S8_FixMoveBack : BOOL;
    LS_S8_FixMoveOut : BOOL;
    SOL_S8_FixMove : BOOL;
    Error_LS_S8_FixMoveBack : BOOL;
    Error_LS_S8_FixMoveOut : BOOL;
    LS_S8_TurnBack : BOOL;
    LS_S8_TurnOut : BOOL;
    SOL_S8_Turn : BOOL;
    Error_LS_S8_TurnBack : BOOL;
    Error_LS_S8_TurnOut : BOOL;
    LS_S8_ClipBack : BOOL;
    LS_S8_ClipOut : BOOL;
    SOL_S8_Clip : BOOL;
    Error_LS_S8_ClipBack : BOOL;
    Error_LS_S8_ClipOut : BOOL;
END_VAR
//**********************************************************************************************************************
(*Station8*)
//**********************************************************************************************************************
ErrorDouble[0](
	bAutoStatus:=AutoStatus,
	bResetPB:=PB_Reset OR HMIPB_PB_Reset,
	bBackLS:=LS_S8_MoveBack,
	bOutLS:=LS_S8_MoveOut,
	bBackSOL:=SOL_S8_MoveBack,
	bOutSOL:=SOL_S8_MoveOut,
	bErrorStatus_Back=>Error_LS_S8_MoveBack,
	bErrorStatus_Out=>Error_LS_S8_MoveOut);

ErrorSingle[0](
	bAutoStatus:=AutoStatus,
	bResetPB:=PB_Reset OR HMIPB_PB_Reset,
	bBackLS:=LS_S8_UpDownBack,
	bOutLS:=LS_S8_UpDownOut,
	bSOL:=SOL_S8_UpDown,
	bErrorStatus_Back=>Error_LS_S8_UpDownBack,
	bErrorStatus_Out=>Error_LS_S8_UpDownOut);

TON_1(IN:= SOL_S8_VacuumF AND NOT(SNR_S8_VacuumF) ,PT:= t#2s);
IF TON_1.Q THEN
	Error_SNR_S8_VacuumF:=TRUE;
END_IF;

TON_2(IN:= SOL_S8_VacuumR AND NOT(SNR_S8_VacuumR) ,PT:= t#2s);
IF TON_2.Q THEN
	Error_SNR_S8_VacuumR:=TRUE;
END_IF;

IF SystemReadyStatus AND OMRON_FQ2_Error THEN
	Error_OMRON_FQ2_Error:=TRUE;
END_IF;
//節流
ErrorSingle[1](
	bAutoStatus:=AutoStatus,
	bResetPB:=PB_Reset OR HMIPB_PB_Reset,
	bBackLS:=LS_S8_THBack,
	bOutLS:=LS_S8_THOut,
	bSOL:=SOL_S8_TH,
	bErrorStatus_Back=>Error_LS_S8_THBack,
	bErrorStatus_Out=>Error_LS_S8_THOut);
//換卡子
ErrorSingle[2](
	bAutoStatus:=AutoStatus,
	bResetPB:=PB_Reset OR HMIPB_PB_Reset,
	bBackLS:=LS_S8_FixBack,
	bOutLS:=LS_S8_FixOut,
	bSOL:=SOL_S8_Fix,
	bErrorStatus_Back=>Error_LS_S8_FixBack,
	bErrorStatus_Out=>Error_LS_S8_FixOut);
ErrorSingle[3](
	bAutoStatus:=AutoStatus,
	bResetPB:=PB_Reset OR HMIPB_PB_Reset,
	bBackLS:=LS_S8_FixMoveBack,
	bOutLS:=LS_S8_FixMoveOut,
	bSOL:=SOL_S8_FixMove,
	bErrorStatus_Back=>Error_LS_S8_FixMoveBack,
	bErrorStatus_Out=>Error_LS_S8_FixMoveOut);
ErrorSingle[4](
	bAutoStatus:=AutoStatus,
	bResetPB:=PB_Reset OR HMIPB_PB_Reset,
	bBackLS:=LS_S8_TurnBack,
	bOutLS:=LS_S8_TurnOut,
	bSOL:=SOL_S8_Turn,
	bErrorStatus_Back=>Error_LS_S8_TurnBack,
	bErrorStatus_Out=>Error_LS_S8_TurnOut);
ErrorSingle[5](
	bAutoStatus:=AutoStatus,
	bResetPB:=PB_Reset OR HMIPB_PB_Reset,
	bBackLS:=LS_S8_ClipBack,
	bOutLS:=LS_S8_ClipOut,
	bSOL:=SOL_S8_Clip,
	bErrorStatus_Back=>Error_LS_S8_ClipBack,
	bErrorStatus_Out=>Error_LS_S8_ClipOut);
//異常
ErrorStatus[8]:=
Error_LS_S8_MoveBack OR
Error_LS_S8_MoveBack OR
Error_LS_S8_UpDownBack OR
Error_LS_S8_UpDownOut OR
Error_SNR_S8_VacuumF OR
Error_SNR_S8_VacuumR OR
Error_OMRON_FQ2_Error;

ErrorStatus_TH[8]:=
Error_LS_S8_THBack OR
Error_LS_S8_THOut;

ErrorStatus_S8_Fix:=
Error_LS_S8_FixBack OR
Error_LS_S8_FixOut OR
Error_LS_S8_FixMoveBack OR
Error_LS_S8_FixMoveOut OR
Error_LS_S8_TurnBack OR
Error_LS_S8_TurnOut OR
Error_LS_S8_ClipBack OR
Error_LS_S8_ClipOut;
//RESET
IF PB_Reset OR HMIPB_PB_Reset THEN
	Error_SNR_S8_VacuumF:=FALSE;
	Error_SNR_S8_VacuumR:=FALSE;
	Error_OMRON_FQ2_Error:=FALSE;
END_IF;
END_PROGRAM

PROGRAM prError_S10
VAR
    ErrorDouble : ARRAY[0..9] of fbErrorDouble;
    ErrorSingle : ARRAY[0..9] of fbErrorSingle;
END_VAR
VAR_EXTERNAL
    AutoStatus : BOOL;
    PB_Reset : BOOL;
    HMIPB_PB_Reset : BOOL;
    LS_S10_MoveBack : BOOL;
    LS_S10_MoveOut : BOOL;
    SOL_S10_MoveBack : BOOL;
    SOL_S10_MoveOut : BOOL;
    Error_LS_S10_MoveBack : BOOL;
    Error_LS_S10_MoveOut : BOOL;
    LS_S10_UpDownBack : BOOL;
    LS_S10_UpDownOut : BOOL;
    SOL_S10_UpDown : BOOL;
    Error_LS_S10_UpDownBack : BOOL;
    Error_LS_S10_UpDownOut : BOOL;
    ErrorStatus : ARRAY[0..19] OF BOOL;
    ErrorStatus_TH : ARRAY[0..19] OF BOOL;
    LS_S10_THBack : BOOL;
    LS_S10_THOut : BOOL;
    SOL_S10_TH : BOOL;
    Error_LS_S10_THBack : BOOL;
    Error_LS_S10_THOut : BOOL;
    LS_S10_ClipFBack : BOOL;
    LS_S10_ClipFOut : BOOL;
    SOL_S10_ClipF : BOOL;
    Error_LS_S10_ClipFBack : BOOL;
    Error_LS_S10_ClipFOut : BOOL;
    LS_S10_ClipRBack : BOOL;
    LS_S10_ClipROut : BOOL;
    SOL_S10_ClipR : BOOL;
    Error_LS_S10_ClipRBack : BOOL;
    Error_LS_S10_ClipROut : BOOL;
END_VAR
//**********************************************************************************************************************
(*Station10*)
//**********************************************************************************************************************
ErrorDouble[0](
	bAutoStatus:=AutoStatus,
	bResetPB:=PB_Reset OR HMIPB_PB_Reset,
	bBackLS:=LS_S10_MoveBack,
	bOutLS:=LS_S10_MoveOut,
	bBackSOL:=SOL_S10_MoveBack,
	bOutSOL:=SOL_S10_MoveOut,
	bErrorStatus_Back=>Error_LS_S10_MoveBack,
	bErrorStatus_Out=>Error_LS_S10_MoveOut);

ErrorSingle[0](
	bAutoStatus:=AutoStatus,
	bResetPB:=PB_Reset OR HMIPB_PB_Reset,
	bBackLS:=LS_S10_UpDownBack,
	bOutLS:=LS_S10_UpDownOut,
	bSOL:=SOL_S10_UpDown,
	bErrorStatus_Back=>Error_LS_S10_UpDownBack,
	bErrorStatus_Out=>Error_LS_S10_UpDownOut);

ErrorSingle[1](
	bAutoStatus:=AutoStatus,
	bResetPB:=PB_Reset OR HMIPB_PB_Reset,
	bBackLS:=LS_S10_ClipFBack,
	bOutLS:=LS_S10_ClipFOut,
	bSOL:=SOL_S10_ClipF,
	bErrorStatus_Back=>Error_LS_S10_ClipFBack,
	bErrorStatus_Out=>Error_LS_S10_ClipFOut);

ErrorSingle[2](
	bAutoStatus:=AutoStatus,
	bResetPB:=PB_Reset OR HMIPB_PB_Reset,
	bBackLS:=LS_S10_ClipRBack,
	bOutLS:=LS_S10_ClipROut,
	bSOL:=SOL_S10_ClipR,
	bErrorStatus_Back=>Error_LS_S10_ClipRBack,
	bErrorStatus_Out=>Error_LS_S10_ClipROut);
//節流
ErrorSingle[3](
	bAutoStatus:=AutoStatus,
	bResetPB:=PB_Reset OR HMIPB_PB_Reset,
	bBackLS:=LS_S10_THBack,
	bOutLS:=LS_S10_THOut,
	bSOL:=SOL_S10_TH,
	bErrorStatus_Back=>Error_LS_S10_THBack,
	bErrorStatus_Out=>Error_LS_S10_THOut);

//異常
ErrorStatus[10]:=
Error_LS_S10_MoveBack OR
Error_LS_S10_MoveBack OR
Error_LS_S10_UpDownBack OR
Error_LS_S10_UpDownOut OR
Error_LS_S10_ClipFBack OR
Error_LS_S10_ClipFOut OR
Error_LS_S10_ClipRBack OR
Error_LS_S10_ClipROut;

ErrorStatus_TH[10]:=
Error_LS_S10_THBack OR
Error_LS_S10_THOut;
END_PROGRAM

PROGRAM prError_S11
VAR
    ErrorSingle : ARRAY[0..1] of fbErrorSingle;
END_VAR
VAR_EXTERNAL
    AutoStatus : BOOL;
    PB_Reset : BOOL;
    HMIPB_PB_Reset : BOOL;
    LS_S11_UpDownBack : BOOL;
    LS_S11_UpDownOut : BOOL;
    SOL_S11_UpDown : BOOL;
    Error_LS_S11_UpDownBack : BOOL;
    Error_LS_S11_UpDownOut : BOOL;
    ErrorStatus : ARRAY[0..19] OF BOOL;
END_VAR
//**********************************************************************************************************************
(*Station11*)
//**********************************************************************************************************************
ErrorSingle[0](
	bAutoStatus:=AutoStatus,
	bResetPB:=PB_Reset OR HMIPB_PB_Reset,
	bBackLS:=LS_S11_UpDownBack,
	bOutLS:=LS_S11_UpDownOut,
	bSOL:=SOL_S11_UpDown,
	bErrorStatus_Back=>Error_LS_S11_UpDownBack,
	bErrorStatus_Out=>Error_LS_S11_UpDownOut);

ErrorStatus[11]:=
Error_LS_S11_UpDownBack OR
Error_LS_S11_UpDownOut;
END_PROGRAM

PROGRAM prError_S13
VAR
    ErrorSingle : ARRAY[0..1] of fbErrorSingle;
END_VAR
VAR_EXTERNAL
    AutoStatus : BOOL;
    PB_Reset : BOOL;
    HMIPB_PB_Reset : BOOL;
    LS_S13_UpDownBack : BOOL;
    LS_S13_UpDownOut : BOOL;
    SOL_S13_UpDown : BOOL;
    Error_LS_S13_UpDownBack : BOOL;
    Error_LS_S13_UpDownOut : BOOL;
    ErrorStatus : ARRAY[0..19] OF BOOL;
END_VAR
//**********************************************************************************************************************
(*Station13*)
//**********************************************************************************************************************
ErrorSingle[0](
	bAutoStatus:=AutoStatus,
	bResetPB:=PB_Reset OR HMIPB_PB_Reset,
	bBackLS:=LS_S13_UpDownBack,
	bOutLS:=LS_S13_UpDownOut,
	bSOL:=SOL_S13_UpDown,
	bErrorStatus_Back=>Error_LS_S13_UpDownBack,
	bErrorStatus_Out=>Error_LS_S13_UpDownOut);

ErrorStatus[13]:=
Error_LS_S13_UpDownBack OR
Error_LS_S13_UpDownOut;
END_PROGRAM

PROGRAM prError_S15
VAR
    ErrorSingle : ARRAY[0..1] of fbErrorSingle;
END_VAR
VAR_EXTERNAL
    AutoStatus : BOOL;
    PB_Reset : BOOL;
    HMIPB_PB_Reset : BOOL;
    LS_S15_UpDownBack : BOOL;
    LS_S15_UpDownOut : BOOL;
    SOL_S15_UpDown : BOOL;
    Error_LS_S15_UpDownBack : BOOL;
    Error_LS_S15_UpDownOut : BOOL;
    ErrorStatus : ARRAY[0..19] OF BOOL;
END_VAR
//**********************************************************************************************************************
(*Station15*)
//**********************************************************************************************************************
ErrorSingle[0](
	bAutoStatus:=AutoStatus,
	bResetPB:=PB_Reset OR HMIPB_PB_Reset,
	bBackLS:=LS_S15_UpDownBack,
	bOutLS:=LS_S15_UpDownOut,
	bSOL:=SOL_S15_UpDown,
	bErrorStatus_Back=>Error_LS_S15_UpDownBack,
	bErrorStatus_Out=>Error_LS_S15_UpDownOut);

ErrorStatus[15]:=
Error_LS_S15_UpDownBack OR
Error_LS_S15_UpDownOut;
END_PROGRAM

PROGRAM prStation1
VAR
    AutoFlow : INT;
    Rtrig_test : R_TRIG;
    TON_CT : TON;
END_VAR
VAR_EXTERNAL
    IndexData : ARRAY[0..19] OF stIndexData;
    DisablePB : ARRAY[0..19] OF BOOL;
    TestPB : ARRAY[0..19] OF BOOL;
    SystemReadyStatus : BOOL;
    AutoStatus : BOOL;
    ErrorStatus : ARRAY[0..19] OF BOOL;
    Error_PB_EStop : BOOL;
    YAMAHA_Load_Start : BOOL;
    MachineRunStatus : BOOL;
    YAMAHA_Load_Finish : BOOL;
    CycleTime : ARRAY[0..19] OF DINT;
    BatchIndexCount : DINT;
END_VAR
(*
程序名稱:第1站上料流程
作者:蔡相偉
版本,日期,版本資訊:
1.0.0		2017/11/21		初始版本
PowerOn=0
Idle=1
上料開始=2
上料完成=3
*)
//本站狀態判斷
IF IndexData[1].OKFlag[1]
	OR IndexData[1].NGFlag[1] THEN
	IndexData[1].FinishFlag[1]:=TRUE;
END_IF;
(*
//前站狀態判斷
IF NOT(IndexData[10].FinishFlag[9]
	AND IndexData[10].OKFlag[9]
	AND NOT(IndexData[10].NGFlag[9])) THEN
	IndexData[10].NGFlag[10]:=TRUE;
END_IF;
*)
//本站關閉判斷
IF DisablePB[1] AND NOT(IndexData[1].FinishFlag[1]) THEN
	IndexData[1].NGFlag[1]:=TRUE;
END_IF;

Rtrig_test(CLK:=TestPB[1]);
//PowerOn=0
IF NOT(SystemReadyStatus AND AutoStatus AND NOT(ErrorStatus[1]) AND NOT(Error_PB_EStop)) THEN
	Autoflow:=0;
END_IF;

//Idle=1
IF AutoFlow=0 AND SystemReadyStatus AND AutoStatus AND NOT(ErrorStatus[1]) AND NOT(Error_PB_EStop) THEN
	AutoFlow:=1;
END_IF;

IF AutoFlow=3 AND NOT(YAMAHA_Load_Start) AND IndexData[1].FinishFlag[1] THEN
	AutoFlow:=1;
END_IF;

//上料開始=2
IF Autoflow=1
	AND AutoStatus
	AND NOT(DisablePB[1])
	AND (MachineRunStatus AND NOT(IndexData[1].FinishFlag[1]) OR Rtrig_test.Q) THEN
	Autoflow:=2;
END_IF;
IF AutoFlow=2 THEN
	YAMAHA_Load_Start:=TRUE;
END_IF;
IF YAMAHA_Load_Finish OR AutoFlow=0 THEN
	YAMAHA_Load_Start:=FALSE;
END_IF;

//上料完成=3
IF AutoFlow=2 AND (YAMAHA_Load_Finish) THEN
	BatchIndexCount:=BatchIndexCount+1;
	AutoFlow:=3;
END_IF;
IF AutoFlow=3 THEN
	IndexData[1].OKFlag[1]:=TRUE;
END_IF;

//*************************************************************************
//Cycle Time
//*************************************************************************
TON_CT(In:=AutoFlow>1, PT:=t#500s);
CycleTime[1]:=LINT_TO_DINT(TimeToSec( TON_CT.ET));
END_PROGRAM

PROGRAM prStation1_Robot
VAR
    R_TRIG1 : R_TRIG;
    R_TRIG2 : R_TRIG;
    R_TRIG3 : R_TRIG;
END_VAR
VAR_EXTERNAL
    HMIPB_YAMAHA_Unload_OKStart : BOOL;
    YAMAHA_Unload_OKStart : BOOL;
    YAMAHA_Unload_NGStart : BOOL;
    HMIPB_YAMAHA_Unload_NGStart : BOOL;
    YAMAHA_Load_Start : BOOL;
    HMIPB_YAMAHA_Load_Start : BOOL;
    YAMAHA_UnLoad_Ready : BOOL;
    HMIPB_YAMAHA_UnLoad_Ready : BOOL;
    HMIPB_YAMAHA_Load_Ready : BOOL;
    YAMAHA_Load_Ready : BOOL;
    HMIPB_YAMAHA_Unload_ChangePanelStart : BOOL;
    YAMAHA_Unload_ChangePanelStart : BOOL;
    HMIPB_YAMAHA_Load_ChangePanelStart : BOOL;
    YAMAHA_Load_ChangePanelStart : BOOL;
    HMIPB_YAMAHA_ORG : BOOL;
    YAMAHA_ORG : BOOL;
    HMIPB_YAMAHA_S_Enable : BOOL;
    YAMAHA_S_Enable : BOOL;
    HMIPB_YAMAHA_S_Control : BOOL;
    YAMAHA_S_Control : BOOL;
    HMIPB_YAMAHA_S_Stop : BOOL;
    YAMAHA_S_Stop : BOOL;
    HMIPB_YAMAHA_S_AutoRun : BOOL;
    YAMAHA_S_AutoRun : BOOL;
    HMIPB_YAMAHA_S_INCHome : BOOL;
    YAMAHA_S_INCHome : BOOL;
    HMIPB_YAMAHA_S_ProgramReset : BOOL;
    YAMAHA_S_ProgramReset : BOOL;
    HMIPB_YAMAHA_S_AlarmReset : BOOL;
    YAMAHA_S_AlarmReset : BOOL;
    HMIPB_YAMAHA_S_ABSHome : BOOL;
    YAMAHA_S_ABSHome : BOOL;
    PB_EStop : BOOL;
    SNR_S1_Door1 : BOOL;
    SNR_S1_Door2 : BOOL;
    SNR_S1_Door3 : BOOL;
    SNR_S1_Door4 : BOOL;
    SystemReadyStatus : BOOL;
    YAMAHA_S_State_CPUOK : BOOL;
    YAMAHA_S_State_Enable : BOOL;
    Error_PB_EStop : BOOL;
    Error_LS_Door : BOOL;
    YAMAHA_S_State_Homed : BOOL;
    YAMAHA_S_State_ProgramReset : BOOL;
    YAMAHA_S_State_RobotProgramRun : BOOL;
END_VAR
//Define
YAMAHA_Unload_OKStart:=HMIPB_YAMAHA_Unload_OKStart;
YAMAHA_Unload_NGStart:=HMIPB_YAMAHA_Unload_NGStart;
YAMAHA_Load_Start:=HMIPB_YAMAHA_Load_Start;
//YAMAHA_UnLoad_Ready:=HMIPB_YAMAHA_UnLoad_Ready;
//YAMAHA_Load_Ready:=HMIPB_YAMAHA_Load_Ready;
YAMAHA_S_Control:=HMIPB_YAMAHA_S_Control;
YAMAHA_S_AutoRun:=HMIPB_YAMAHA_S_AutoRun;
YAMAHA_S_INCHome:=HMIPB_YAMAHA_S_INCHome;
YAMAHA_S_ProgramReset:=HMIPB_YAMAHA_S_ProgramReset;
YAMAHA_S_AlarmReset:=HMIPB_YAMAHA_S_AlarmReset;
YAMAHA_S_ABSHome:=HMIPB_YAMAHA_S_ABSHome;

//********************************************************************************************************
//ROBOT伺服ON流程
//********************************************************************************************************
R_TRIG1(Clk:=(SystemReadyStatus AND YAMAHA_S_State_CPUOK) OR HMIPB_YAMAHA_S_Enable);
IF R_TRIG1.Q THEN
	YAMAHA_S_Enable:=TRUE;
END_IF;
IF YAMAHA_S_State_Enable THEN
	YAMAHA_S_Enable:=FALSE;
END_IF;
//********************************************************************************************************
//STOP ON
//********************************************************************************************************
YAMAHA_S_Stop:=
HMIPB_YAMAHA_S_Stop AND
NOT(Error_PB_EStop) AND
NOT(Error_LS_Door);
//********************************************************************************************************
//程序復位和執行
//********************************************************************************************************
R_TRIG2(Clk:=YAMAHA_S_State_Homed AND YAMAHA_S_State_Enable AND YAMAHA_S_Stop AND HMIPB_YAMAHA_S_ProgramReset);
R_TRIG3(Clk:=YAMAHA_S_State_Homed AND YAMAHA_S_State_Enable AND YAMAHA_S_Stop AND YAMAHA_S_State_ProgramReset AND HMIPB_YAMAHA_S_AutoRun);
IF R_TRIG2.Q THEN
	YAMAHA_S_ProgramReset:=TRUE;
END_IF;
IF YAMAHA_S_State_ProgramReset THEN
	YAMAHA_S_ProgramReset:=FALSE;
END_IF;
IF R_TRIG3.Q THEN
	YAMAHA_S_AutoRun:=TRUE;
END_IF;
IF YAMAHA_S_State_RobotProgramRun AND NOT(YAMAHA_S_State_ProgramReset) THEN
	YAMAHA_S_AutoRun:=FALSE;
END_IF;
END_PROGRAM

PROGRAM prStation1_PanelLoad
VAR
    Autoflow : INT;
    Initflow : INT;
    interlockback : ARRAY[0..2] OF BOOL;
    interlockout : ARRAY[0..2] OF BOOL;
    solStatus : ARRAY[0..2] OF BOOL;
    R_TRIG_1 : ARRAY[0..2] OF R_TRIG;
    F_TRIG_1 : F_TRIG;
    ErrorLS : BOOL;
    StartFlag : BOOL;
    TON_1 : TON;
    TON_2 : TON;
    TON_3 : TON;
    Rtrig_test : R_TRIG;
END_VAR
VAR_EXTERNAL
    HMIPB_SOL_S1_Load_PanelUpDown1Back : BOOL;
    SOL_S1_Load_PanelUpDown1Back : BOOL;
    SOL_S1_Load_PanelUpDown1Out : BOOL;
    LS_S1_Load_PanelUpDown1Back : BOOL;
    HMIPB_SOL_S1_Load_PanelUpDown1Out : BOOL;
    AutoStatus : BOOL;
    LS_S1_Load_PanelUpDown1Out : BOOL;
    HMIPB_SOL_S1_Load_PanelUpDown2Back : BOOL;
    SOL_S1_Load_PanelUpDown2Back : BOOL;
    SOL_S1_Load_PanelUpDown2Out : BOOL;
    LS_S1_Load_PanelUpDown2Back : BOOL;
    HMIPB_SOL_S1_Load_PanelUpDown2Out : BOOL;
    LS_S1_Load_PanelUpDown2Out : BOOL;
    HMIPB_SOL_S1_Load_PanelClip : BOOL;
    SOL_S1_Load_PanelClip : BOOL;
    SystemReadyStatus : BOOL;
    ErrorStatus : ARRAY[0..19] OF BOOL;
    Error_PB_EStop : BOOL;
    SNR_S1_Load_PanelFeed : BOOL;
    LS_S1_Load_PanelClip1Out : BOOL;
    LS_S1_Load_PanelClip2Out : BOOL;
    LS_S1_Load_PanelClip2Back : BOOL;
    LS_S1_Load_PanelClip1Back : BOOL;
    RY_S1_Load_VariableSpeedMotor : BOOL;
    Error_LS_S1_Load_PanelUpDown1Back : BOOL;
    Error_LS_S1_Load_PanelUpDown1Out : BOOL;
    Error_LS_S1_Load_PanelUpDown2Back : BOOL;
    Error_LS_S1_Load_PanelUpDown2Out : BOOL;
    Error_LS_S1_Load_PanelClip1Back : BOOL;
    Error_LS_S1_Load_PanelClip1Out : BOOL;
    Error_LS_S1_Load_PanelClip2Back : BOOL;
    Error_LS_S1_Load_PanelClip2Out : BOOL;
    ErrorStatus_S1_Load : BOOL;
    Error_SNR_S1_Load_PanelFeed : BOOL;
    PB_Reset : BOOL;
    HMIPB_PB_Reset : BOOL;
    StepMode : BOOL;
END_VAR
(*
程序名稱: Panel LOAD程序
作者:蔡相偉
版本,日期,版本資訊:
1.0.0		2017/11/16		初始版本

PowerOn=0
Idle=1
Panel出盤程序開始=10
第1段,第2段出=2
夾持出=3
第2段回=4
夾持回=5
第1段回=6
第1段到回=7
*)
//***************************************************************************************************************
//Define
ErrorLS:=ErrorStatus_S1_Load;
StartFlag:=TON_1.Q;
TON_1(In:=NOT(SNR_S1_Load_PanelFeed) AND NOT(RY_S1_Load_VariableSpeedMotor), PT:=t#5s);
//PowerOn=0
IF NOT(SystemReadyStatus AND NOT(ErrorLS) AND  NOT(Error_PB_Estop) AND AutoStatus) THEN
	Autoflow:=0;
END_IF;

//Idle=1
IF AutoFlow=0 AND SystemReadyStatus AND NOT(ErrorLS) AND  NOT(Error_PB_Estop) AND AutoStatus THEN
	AutoFlow:=1;
END_IF;

IF Autoflow=7 AND (Error_SNR_S1_Load_PanelFeed OR SNR_S1_Load_PanelFeed) THEN
	Autoflow:=1;
END_IF;

//第1段,第2段出=2
IF Autoflow=1 AND NOT(Error_SNR_S1_Load_PanelFeed) AND StartFlag THEN
	Autoflow:=2;
END_IF;

//承盤夾持出=3
IF Autoflow=2 AND LS_S1_Load_PanelUpDown1Out AND LS_S1_Load_PanelUpDown2Out AND (Rtrig_test.Q OR NOT(StepMode)) THEN
	Autoflow:=3;
END_IF;
TON_2(In:= Autoflow=3 AND LS_S1_Load_PanelClip1Out AND LS_S1_Load_PanelClip2Out , PT:=t#300ms);

//第2段回=4
IF Autoflow=3 AND TON_2.Q AND (Rtrig_test.Q OR NOT(StepMode)) THEN
	Autoflow:=4;
END_IF;
TON_3(In:=Autoflow=4 AND LS_S1_Load_PanelUpDown2Back, PT:=t#300ms);

//承盤夾持回=5
IF Autoflow=4 AND TON_3.Q AND (Rtrig_test.Q OR NOT(StepMode)) THEN
	Autoflow:=5;
END_IF;

//第1段回=6
IF Autoflow=5 AND  LS_S1_Load_PanelClip1Back AND LS_S1_Load_PanelClip2Back AND (Rtrig_test.Q OR NOT(StepMode)) THEN
	Autoflow:=6;
END_IF;

//第1段到回=7
IF Autoflow=6 AND  LS_S1_Load_PanelUpDown1Back AND (Rtrig_test.Q OR NOT(StepMode)) THEN
	Autoflow:=7;
END_IF;
IF Autoflow=7 AND NOT(SNR_S1_Load_PanelFeed) THEN
	Error_SNR_S1_Load_PanelFeed:=TRUE;
END_IF;

//***************************************************************************************************************
//下夾板出盤下降第1段回電磁閥
interlockback[0]:=TRUE;
IF ((HMIPB_SOL_S1_Load_PanelUpDown1Back AND NOT(AutoStatus)) OR Autoflow=6 OR Initflow=6) AND interlockback[0] THEN
	SOL_S1_Load_PanelUpDown1Back:=TRUE;
	SOL_S1_Load_PanelUpDown1Out:=FALSE;
END_IF;
IF LS_S1_Load_PanelUpDown1Back THEN
	SOL_S1_Load_PanelUpDown1Back:=FALSE;
END_IF;

//下夾板出盤下降第1段出電磁閥
interlockout[0]:=TRUE;
IF ((HMIPB_SOL_S1_Load_PanelUpDown1Out AND NOT(AutoStatus)) OR Autoflow=2) AND interlockout[0] THEN
	SOL_S1_Load_PanelUpDown1Back:=FALSE;
	SOL_S1_Load_PanelUpDown1Out:=TRUE;
END_IF;
IF LS_S1_Load_PanelUpDown1Out THEN
	SOL_S1_Load_PanelUpDown1Out:=FALSE;
END_IF;
//***************************************************************************************************************
//下夾板出盤下降第2段回電磁閥
interlockback[1]:=TRUE;
IF ((HMIPB_SOL_S1_Load_PanelUpDown2Back AND NOT(AutoStatus)) OR Autoflow=4 OR Initflow=4) AND interlockback[1] THEN
	SOL_S1_Load_PanelUpDown2Back:=TRUE;
	SOL_S1_Load_PanelUpDown2Out:=FALSE;
END_IF;
IF LS_S1_Load_PanelUpDown2Back THEN
	SOL_S1_Load_PanelUpDown2Back:=FALSE;
END_IF;

//下夾板出盤下降第2段出電磁閥
interlockout[1]:=LS_S1_Load_PanelUpDown1Out AND NOT(SNR_S1_Load_PanelFeed);
IF ((HMIPB_SOL_S1_Load_PanelUpDown2Out AND NOT(AutoStatus)) OR Autoflow=2) AND interlockout[1] THEN
	SOL_S1_Load_PanelUpDown2Back:=FALSE;
	SOL_S1_Load_PanelUpDown2Out:=TRUE;
END_IF;
IF LS_S1_Load_PanelUpDown2Out THEN
	SOL_S1_Load_PanelUpDown2Out:=FALSE;
END_IF;
//***************************************************************************************************************
(*下夾板出盤承載電磁閥*)
R_TRIG_1[2](CLK:=HMIPB_SOL_S1_Load_PanelClip AND NOT(AutoStatus));
interlockback[2]:=TRUE;
interlockout[2]:=LS_S1_Load_PanelUpDown1Out;
(*SET*)
IF ((R_TRIG_1[2].Q AND NOT(solStatus[2])) OR Autoflow=3) AND interlockout[2] THEN
	SOL_S1_Load_PanelClip:=TRUE;
END_IF;
(*RESET*)
IF ((R_TRIG_1[2].Q AND (solStatus[2])) OR Autoflow=5 OR Initflow=5) AND interlockback[2] THEN
	SOL_S1_Load_PanelClip:=FALSE;
END_IF;
(*STATUS*)
solStatus[2]:=SOL_S1_Load_PanelClip;

//***************************************************************************************************************
(*
程序名稱: Panel LOAD RESET程序
作者:蔡相偉
版本,日期,版本資訊:
1.0.0		2017/11/16		初始版本

PowerOn=0
Idle=1
第2段回=4
夾持回=5
第1段回=6

//***************************************************************************************************************
//PowerOn=0
IF NOT(SystemReadyStatus) THEN
	Initflow:=0;
END_IF;

//Idle=1
IF Initflow=0 AND SystemReadyStatus THEN
	Initflow:=1;
END_IF;

IF Initflow=6 AND LS_S1_Load_PanelUpDown1Back THEN
	Initflow:=1;
END_IF;

